# B&R Automation Studio project ControlPLC_DataDistribution (part 2)

### IoMap.iom - 5PC900_TS17_02/IoMap.iom
```iecst
VAR_CONFIG
	::VFLCR_Ope0:IO.raw.oSystemControl AT %QD."VF-LCR".SYSTEM_CONTROL_I2004Out;
	::VFLCR_Ope0:IO.ao.SelectedPrintNumber AT %QD."VF-LCR".SELECTED_PRINT_NUMBER_I200BOut;
	::VFLCR_Ope0:IO.ao.SelectedLayerNumber AT %QD."VF-LCR".SELECTED_LAYER_NUMBER_I200COut;
	::VFLCR_Ope0:IO.ao.SelectedBuildLayout AT %QD."VF-LCR".SELECTED_BUILD_LAYOUT_I200AOut;
	::VFLCR_Ope0:IO.ao.PLCHeartbeat AT %QD."VF-LCR".PLC_HEARTBEAT_I2003Out;
	::VFLCR_Ope0:IO.raw.oOperationControl AT %QD."VF-LCR".OPERATION_CONTROL_I2005Out;
	::VFLCR_Ope0:IO.raw.oManualLaserOperation AT %QD."VF-LCR".MANUAL_LASER_OPERATION_I200EOut;
	::VFLCR_Ope0:IO.raw.oManualLaserCurrentSetpoint AT %QD."VF-LCR".MANUAL_LASER_CURRENT_SETPOINT_I200FOut;
	::VFLCR_Ope0:IO.raw.oLaserEnable AT %QD."VF-LCR".LASER_ENABLE_I2008Out;
	::VFLCR_Ope0:IO.raw.oEnableLaserMainPower AT %QD."VF-LCR".LASER_REMOTE_START_I2010Out;
	::VFLCR_Ope0:IO.raw.oEnableLaserEmission AT %QD."VF-LCR".LASER_EMISSION_CONTROL_I2012Out;
	::VFLCR_Ope0:IO.raw.oEnableGuideLaser AT %QD."VF-LCR".GUIDE_LASER_CONTROL_I2011Out;
	::VFLCR_Ope0:IO.raw.oResetLaserErrors AT %QD."VF-LCR".LASER_RESET_I2013Out;
	::VFLCR_Ope0:IO.di.PowerlinkModuleOK AT %IX."VF-LCR".ModuleOk;
	::VFLCR_Ope0:IO.ai.DMACurrentTrajectory[0] AT %ID."VF-LCR".Entry_I201B_S01;
	::VFLCR_Ope0:IO.raw.iLaserFatalError AT %ID."VF-LCR".SYSTEM_ERROR_I2018;
	::VFLCR_Ope0:IO.raw.iSystemStatus AT %ID."VF-LCR".SYSTEM_STATUS_I2006;
	::VFLCR_Ope0:IO.ai.SystemHeartbeat AT %ID."VF-LCR".SYSTEM_HEARTBEAT_I2002;
	::VFLCR_Ope0:IO.raw.iSoftwareRevision AT %ID."VF-LCR".SOFTWARE_REVISION_I201D;
	::VFLCR_Ope0:IO.raw.iOperationStatus AT %ID."VF-LCR".OPERATION_STATUS_I2007;
	::VFLCR_Ope0:IO.raw.iManualModeLaserPower AT %ID."VF-LCR".LASER_POWER_MONITOR_I2019;
	::VFLCR_Ope0:IO.ai.LUTFiles_CalibrationID AT %ID."VF-LCR".LUT_LOAD_STATUS_I2009;
	::VFLCR_Ope0:IO.raw.iLaserWatchdogError AT %ID."VF-LCR".LASER_WATCHDOG_ERROR_I201E;
	::VFLCR_Ope0:IO.raw.iLaserEmissionEnabled AT %ID."VF-LCR".LASER_EMISSION_ON_I2017;
	::VFLCR_Ope0:IO.raw.iLaserControlPowerEnabled AT %ID."VF-LCR".LASER_CONTROL_SYSTEM_POWERED_ON_I2015;
	::VFLCR_Ope0:IO.raw.iFPGARevision AT %ID."VF-LCR".FPGA_REVISION_I2001;
	::VFLCR_Ope0:IO.ai.DMAStatus[8] AT %ID."VF-LCR".Entry_I201A_S09;
	::VFLCR_Ope0:IO.ai.DMAStatus[7] AT %ID."VF-LCR".Entry_I201A_S08;
	::VFLCR_Ope0:IO.ai.DMAStatus[6] AT %ID."VF-LCR".Entry_I201A_S07;
	::VFLCR_Ope0:IO.ai.DMAStatus[5] AT %ID."VF-LCR".Entry_I201A_S06;
	::VFLCR_Ope0:IO.ai.DMAStatus[4] AT %ID."VF-LCR".Entry_I201A_S05;
	::VFLCR_Ope0:IO.ai.DMAStatus[3] AT %ID."VF-LCR".Entry_I201A_S04;
	::VFLCR_Ope0:IO.ai.DMAStatus[13] AT %ID."VF-LCR".Entry_I201A_S0E;
	::VFLCR_Ope0:IO.ai.DMAStatus[2] AT %ID."VF-LCR".Entry_I201A_S03;
	::VFLCR_Ope0:IO.ai.DMAStatus[19] AT %ID."VF-LCR".Entry_I201A_S14;
	::VFLCR_Ope0:IO.ai.DMAStatus[1] AT %ID."VF-LCR".Entry_I201A_S02;
	::VFLCR_Ope0:IO.ai.DMAStatus[18] AT %ID."VF-LCR".Entry_I201A_S13;
	::VFLCR_Ope0:IO.ai.DMAStatus[17] AT %ID."VF-LCR".Entry_I201A_S12;
	::VFLCR_Ope0:IO.ai.DMAStatus[16] AT %ID."VF-LCR".Entry_I201A_S11;
	::VFLCR_Ope0:IO.ai.DMAStatus[15] AT %ID."VF-LCR".Entry_I201A_S10;
	::VFLCR_Ope0:IO.ai.DMAStatus[14] AT %ID."VF-LCR".Entry_I201A_S0F;
	::VFLCR_Ope0:IO.raw.iLaserMainPowerEnabled AT %ID."VF-LCR".LASER_MAIN_POWER_ON_I2016;
	::VFLCR_Ope0:IO.raw.iLaserReady_Error AT %ID."VF-LCR".LASER_ERROR_READY_I2014;
	::VFLCR_Ope0:IO.ai.DMAStatus[20] AT %ID."VF-LCR".Entry_I201A_S15;
	::VFLCR_Ope0:IO.ai.DMAStatus[12] AT %ID."VF-LCR".Entry_I201A_S0D;
	::VFLCR_Ope0:IO.ai.DMACurrentTrajectory[7] AT %ID."VF-LCR".Entry_I201B_S08;
	::VFLCR_Ope0:IO.ai.DMAStatus[0] AT %ID."VF-LCR".Entry_I201A_S01;
	::VFLCR_Ope0:IO.ai.DMALastPacketPosition[8] AT %ID."VF-LCR".Entry_I201C_S09;
	::VFLCR_Ope0:IO.ai.DMALastPacketPosition[7] AT %ID."VF-LCR".Entry_I201C_S08;
	::VFLCR_Ope0:IO.ai.DMALastPacketPosition[6] AT %ID."VF-LCR".Entry_I201C_S07;
	::VFLCR_Ope0:IO.ai.DMALastPacketPosition[5] AT %ID."VF-LCR".Entry_I201C_S06;
	::VFLCR_Ope0:IO.ai.DMALastPacketPosition[4] AT %ID."VF-LCR".Entry_I201C_S05;
	::VFLCR_Ope0:IO.ai.DMALastPacketPosition[3] AT %ID."VF-LCR".Entry_I201C_S04;
	::VFLCR_Ope0:IO.ai.DMALastPacketPosition[2] AT %ID."VF-LCR".Entry_I201C_S03;
	::VFLCR_Ope0:IO.ai.DMALastPacketPosition[19] AT %ID."VF-LCR".Entry_I201C_S14;
	::VFLCR_Ope0:IO.ai.DMAStatus[9] AT %ID."VF-LCR".Entry_I201A_S0A;
	::VFLCR_Ope0:IO.ai.DMALastPacketPosition[20] AT %ID."VF-LCR".Entry_I201C_S15;
	::VFLCR_Ope0:IO.ai.DMALastPacketPosition[18] AT %ID."VF-LCR".Entry_I201C_S13;
	::VFLCR_Ope0:IO.ai.DMALastPacketPosition[17] AT %ID."VF-LCR".Entry_I201C_S12;
	::VFLCR_Ope0:IO.ai.DMALastPacketPosition[16] AT %ID."VF-LCR".Entry_I201C_S11;
	::VFLCR_Ope0:IO.ai.DMALastPacketPosition[15] AT %ID."VF-LCR".Entry_I201C_S10;
	::VFLCR_Ope0:IO.ai.DMALastPacketPosition[14] AT %ID."VF-LCR".Entry_I201C_S0F;
	::VFLCR_Ope0:IO.ai.DMALastPacketPosition[13] AT %ID."VF-LCR".Entry_I201C_S0E;
	::VFLCR_Ope0:IO.ai.DMALastPacketPosition[12] AT %ID."VF-LCR".Entry_I201C_S0D;
	::VFLCR_Ope0:IO.ai.DMALastPacketPosition[11] AT %ID."VF-LCR".Entry_I201C_S0C;
	::VFLCR_Ope0:IO.ai.DMAStatus[10] AT %ID."VF-LCR".Entry_I201A_S0B;
	::VFLCR_Ope0:IO.ai.DMALastPacketPosition[1] AT %ID."VF-LCR".Entry_I201C_S02;
	::VFLCR_Ope0:IO.ai.DMAStatus[11] AT %ID."VF-LCR".Entry_I201A_S0C;
	::VFLCR_Ope0:IO.ai.DMALastPacketPosition[10] AT %ID."VF-LCR".Entry_I201C_S0B;
	::VFLCR_Ope0:IO.ai.DMALastPacketPosition[0] AT %ID."VF-LCR".Entry_I201C_S01;
	::VFLCR_Ope0:IO.ai.DMACurrentTrajectory[6] AT %ID."VF-LCR".Entry_I201B_S07;
	::VFLCR_Ope0:IO.ai.DMACurrentTrajectory[5] AT %ID."VF-LCR".Entry_I201B_S06;
	::VFLCR_Ope0:IO.ai.DMACurrentTrajectory[4] AT %ID."VF-LCR".Entry_I201B_S05;
	::VFLCR_Ope0:IO.ai.DMACurrentTrajectory[3] AT %ID."VF-LCR".Entry_I201B_S04;
	::VFLCR_Ope0:IO.ai.DMACurrentTrajectory[2] AT %ID."VF-LCR".Entry_I201B_S03;
	::VFLCR_Ope0:IO.ai.DMACurrentTrajectory[20] AT %ID."VF-LCR".Entry_I201B_S15;
	::VFLCR_Ope0:IO.ai.DMACurrentTrajectory[19] AT %ID."VF-LCR".Entry_I201B_S14;
	::VFLCR_Ope0:IO.ai.DMACurrentTrajectory[1] AT %ID."VF-LCR".Entry_I201B_S02;
	::VFLCR_Ope0:IO.ai.DMACurrentTrajectory[18] AT %ID."VF-LCR".Entry_I201B_S13;
	::VFLCR_Ope0:IO.ai.DMALastPacketPosition[9] AT %ID."VF-LCR".Entry_I201C_S0A;
	::VFLCR_Ope0:IO.ai.DMACurrentTrajectory[17] AT %ID."VF-LCR".Entry_I201B_S12;
	::VFLCR_Ope0:IO.ai.DMACurrentTrajectory[15] AT %ID."VF-LCR".Entry_I201B_S10;
	::VFLCR_Ope0:IO.ai.DMACurrentTrajectory[14] AT %ID."VF-LCR".Entry_I201B_S0F;
	::VFLCR_Ope0:IO.ai.DMACurrentTrajectory[13] AT %ID."VF-LCR".Entry_I201B_S0E;
	::VFLCR_Ope0:IO.ai.DMACurrentTrajectory[12] AT %ID."VF-LCR".Entry_I201B_S0D;
	::VFLCR_Ope0:IO.ai.DMACurrentTrajectory[11] AT %ID."VF-LCR".Entry_I201B_S0C;
	::VFLCR_Ope0:IO.ai.DMACurrentTrajectory[10] AT %ID."VF-LCR".Entry_I201B_S0B;
	::VFLCR_Ope0:IO.ai.DMACurrentTrajectory[9] AT %ID."VF-LCR".Entry_I201B_S0A;
	::VFLCR_Ope0:IO.ai.DMACurrentTrajectory[8] AT %ID."VF-LCR".Entry_I201B_S09;
	::VFLCR_Ope0:IO.ai.DMACurrentTrajectory[16] AT %ID."VF-LCR".Entry_I201B_S11;
	::VFLCR_Ope1:IO.raw.oSystemControl AT %QD."VF-LCR1".SYSTEM_CONTROL_I2004Out;
	::VFLCR_Ope1:IO.ao.SelectedPrintNumber AT %QD."VF-LCR1".SELECTED_PRINT_NUMBER_I200BOut;
	::VFLCR_Ope1:IO.ao.SelectedLayerNumber AT %QD."VF-LCR1".SELECTED_LAYER_NUMBER_I200COut;
	::VFLCR_Ope1:IO.ao.SelectedBuildLayout AT %QD."VF-LCR1".SELECTED_BUILD_LAYOUT_I200AOut;
	::VFLCR_Ope1:IO.ao.PLCHeartbeat AT %QD."VF-LCR1".PLC_HEARTBEAT_I2003Out;
	::VFLCR_Ope1:IO.raw.oOperationControl AT %QD."VF-LCR1".OPERATION_CONTROL_I2005Out;
	::VFLCR_Ope1:IO.raw.oManualLaserOperation AT %QD."VF-LCR1".MANUAL_LASER_OPERATION_I200EOut;
	::VFLCR_Ope1:IO.raw.oManualLaserCurrentSetpoint AT %QD."VF-LCR1".MANUAL_LASER_CURRENT_SETPOINT_I200FOut;
	::VFLCR_Ope1:IO.raw.oLaserEnable AT %QD."VF-LCR1".LASER_ENABLE_I2008Out;
	::VFLCR_Ope1:IO.raw.oEnableLaserMainPower AT %QD."VF-LCR1".LASER_REMOTE_START_I2010Out;
	::VFLCR_Ope1:IO.raw.oEnableLaserEmission AT %QD."VF-LCR1".LASER_EMISSION_CONTROL_I2012Out;
	::VFLCR_Ope1:IO.raw.oEnableGuideLaser AT %QD."VF-LCR1".GUIDE_LASER_CONTROL_I2011Out;
	::VFLCR_Ope1:IO.raw.oResetLaserErrors AT %QD."VF-LCR1".LASER_RESET_I2013Out;
	::VFLCR_Ope1:IO.di.PowerlinkModuleOK AT %IX."VF-LCR1".ModuleOk;
	::VFLCR_Ope1:IO.ai.DMACurrentTrajectory[0] AT %ID."VF-LCR1".Entry_I201B_S01;
	::VFLCR_Ope1:IO.raw.iLaserFatalError AT %ID."VF-LCR1".SYSTEM_ERROR_I2018;
	::VFLCR_Ope1:IO.raw.iSystemStatus AT %ID."VF-LCR1".SYSTEM_STATUS_I2006;
	::VFLCR_Ope1:IO.ai.SystemHeartbeat AT %ID."VF-LCR1".SYSTEM_HEARTBEAT_I2002;
	::VFLCR_Ope1:IO.raw.iSoftwareRevision AT %ID."VF-LCR1".SOFTWARE_REVISION_I201D;
	::VFLCR_Ope1:IO.raw.iOperationStatus AT %ID."VF-LCR1".OPERATION_STATUS_I2007;
	::VFLCR_Ope1:IO.raw.iManualModeLaserPower AT %ID."VF-LCR1".LASER_POWER_MONITOR_I2019;
	::VFLCR_Ope1:IO.ai.LUTFiles_CalibrationID AT %ID."VF-LCR1".LUT_LOAD_STATUS_I2009;
	::VFLCR_Ope1:IO.raw.iLaserWatchdogError AT %ID."VF-LCR1".LASER_WATCHDOG_ERROR_I201E;
	::VFLCR_Ope1:IO.raw.iLaserEmissionEnabled AT %ID."VF-LCR1".LASER_EMISSION_ON_I2017;
	::VFLCR_Ope1:IO.raw.iLaserControlPowerEnabled AT %ID."VF-LCR1".LASER_CONTROL_SYSTEM_POWERED_ON_I2015;
	::VFLCR_Ope1:IO.raw.iFPGARevision AT %ID."VF-LCR1".FPGA_REVISION_I2001;
	::VFLCR_Ope1:IO.ai.DMAStatus[8] AT %ID."VF-LCR1".Entry_I201A_S09;
	::VFLCR_Ope1:IO.ai.DMAStatus[7] AT %ID."VF-LCR1".Entry_I201A_S08;
	::VFLCR_Ope1:IO.ai.DMAStatus[6] AT %ID."VF-LCR1".Entry_I201A_S07;
	::VFLCR_Ope1:IO.ai.DMAStatus[5] AT %ID."VF-LCR1".Entry_I201A_S06;
	::VFLCR_Ope1:IO.ai.DMAStatus[4] AT %ID."VF-LCR1".Entry_I201A_S05;
	::VFLCR_Ope1:IO.ai.DMAStatus[3] AT %ID."VF-LCR1".Entry_I201A_S04;
	::VFLCR_Ope1:IO.ai.DMAStatus[13] AT %ID."VF-LCR1".Entry_I201A_S0E;
	::VFLCR_Ope1:IO.ai.DMAStatus[2] AT %ID."VF-LCR1".Entry_I201A_S03;
	::VFLCR_Ope1:IO.ai.DMAStatus[19] AT %ID."VF-LCR1".Entry_I201A_S14;
	::VFLCR_Ope1:IO.ai.DMAStatus[1] AT %ID."VF-LCR1".Entry_I201A_S02;
	::VFLCR_Ope1:IO.ai.DMAStatus[18] AT %ID."VF-LCR1".Entry_I201A_S13;
	::VFLCR_Ope1:IO.ai.DMAStatus[17] AT %ID."VF-LCR1".Entry_I201A_S12;
	::VFLCR_Ope1:IO.ai.DMAStatus[16] AT %ID."VF-LCR1".Entry_I201A_S11;
	::VFLCR_Ope1:IO.ai.DMAStatus[15] AT %ID."VF-LCR1".Entry_I201A_S10;
	::VFLCR_Ope1:IO.ai.DMAStatus[14] AT %ID."VF-LCR1".Entry_I201A_S0F;
	::VFLCR_Ope1:IO.raw.iLaserMainPowerEnabled AT %ID."VF-LCR1".LASER_MAIN_POWER_ON_I2016;
	::VFLCR_Ope1:IO.raw.iLaserReady_Error AT %ID."VF-LCR1".LASER_ERROR_READY_I2014;
	::VFLCR_Ope1:IO.ai.DMAStatus[20] AT %ID."VF-LCR1".Entry_I201A_S15;
	::VFLCR_Ope1:IO.ai.DMAStatus[12] AT %ID."VF-LCR1".Entry_I201A_S0D;
	::VFLCR_Ope1:IO.ai.DMACurrentTrajectory[7] AT %ID."VF-LCR1".Entry_I201B_S08;
	::VFLCR_Ope1:IO.ai.DMAStatus[0] AT %ID."VF-LCR1".Entry_I201A_S01;
	::VFLCR_Ope1:IO.ai.DMALastPacketPosition[8] AT %ID."VF-LCR1".Entry_I201C_S09;
	::VFLCR_Ope1:IO.ai.DMALastPacketPosition[7] AT %ID."VF-LCR1".Entry_I201C_S08;
	::VFLCR_Ope1:IO.ai.DMALastPacketPosition[6] AT %ID."VF-LCR1".Entry_I201C_S07;
	::VFLCR_Ope1:IO.ai.DMALastPacketPosition[5] AT %ID."VF-LCR1".Entry_I201C_S06;
	::VFLCR_Ope1:IO.ai.DMALastPacketPosition[4] AT %ID."VF-LCR1".Entry_I201C_S05;
	::VFLCR_Ope1:IO.ai.DMALastPacketPosition[3] AT %ID."VF-LCR1".Entry_I201C_S04;
	::VFLCR_Ope1:IO.ai.DMALastPacketPosition[2] AT %ID."VF-LCR1".Entry_I201C_S03;
	::VFLCR_Ope1:IO.ai.DMALastPacketPosition[19] AT %ID."VF-LCR1".Entry_I201C_S14;
	::VFLCR_Ope1:IO.ai.DMAStatus[9] AT %ID."VF-LCR1".Entry_I201A_S0A;
	::VFLCR_Ope1:IO.ai.DMALastPacketPosition[20] AT %ID."VF-LCR1".Entry_I201C_S15;
	::VFLCR_Ope1:IO.ai.DMALastPacketPosition[18] AT %ID."VF-LCR1".Entry_I201C_S13;
	::VFLCR_Ope1:IO.ai.DMALastPacketPosition[17] AT %ID."VF-LCR1".Entry_I201C_S12;
	::VFLCR_Ope1:IO.ai.DMALastPacketPosition[16] AT %ID."VF-LCR1".Entry_I201C_S11;
	::VFLCR_Ope1:IO.ai.DMALastPacketPosition[15] AT %ID."VF-LCR1".Entry_I201C_S10;
	::VFLCR_Ope1:IO.ai.DMALastPacketPosition[14] AT %ID."VF-LCR1".Entry_I201C_S0F;
	::VFLCR_Ope1:IO.ai.DMALastPacketPosition[13] AT %ID."VF-LCR1".Entry_I201C_S0E;
	::VFLCR_Ope1:IO.ai.DMALastPacketPosition[12] AT %ID."VF-LCR1".Entry_I201C_S0D;
	::VFLCR_Ope1:IO.ai.DMALastPacketPosition[11] AT %ID."VF-LCR1".Entry_I201C_S0C;
	::VFLCR_Ope1:IO.ai.DMAStatus[10] AT %ID."VF-LCR1".Entry_I201A_S0B;
	::VFLCR_Ope1:IO.ai.DMALastPacketPosition[1] AT %ID."VF-LCR1".Entry_I201C_S02;
	::VFLCR_Ope1:IO.ai.DMAStatus[11] AT %ID."VF-LCR1".Entry_I201A_S0C;
	::VFLCR_Ope1:IO.ai.DMALastPacketPosition[10] AT %ID."VF-LCR1".Entry_I201C_S0B;
	::VFLCR_Ope1:IO.ai.DMALastPacketPosition[0] AT %ID."VF-LCR1".Entry_I201C_S01;
	::VFLCR_Ope1:IO.ai.DMACurrentTrajectory[6] AT %ID."VF-LCR1".Entry_I201B_S07;
	::VFLCR_Ope1:IO.ai.DMACurrentTrajectory[5] AT %ID."VF-LCR1".Entry_I201B_S06;
	::VFLCR_Ope1:IO.ai.DMACurrentTrajectory[4] AT %ID."VF-LCR1".Entry_I201B_S05;
	::VFLCR_Ope1:IO.ai.DMACurrentTrajectory[3] AT %ID."VF-LCR1".Entry_I201B_S04;
	::VFLCR_Ope1:IO.ai.DMACurrentTrajectory[2] AT %ID."VF-LCR1".Entry_I201B_S03;
	::VFLCR_Ope1:IO.ai.DMACurrentTrajectory[20] AT %ID."VF-LCR1".Entry_I201B_S15;
	::VFLCR_Ope1:IO.ai.DMACurrentTrajectory[19] AT %ID."VF-LCR1".Entry_I201B_S14;
	::VFLCR_Ope1:IO.ai.DMACurrentTrajectory[1] AT %ID."VF-LCR1".Entry_I201B_S02;
	::VFLCR_Ope1:IO.ai.DMACurrentTrajectory[18] AT %ID."VF-LCR1".Entry_I201B_S13;
	::VFLCR_Ope1:IO.ai.DMALastPacketPosition[9] AT %ID."VF-LCR1".Entry_I201C_S0A;
	::VFLCR_Ope1:IO.ai.DMACurrentTrajectory[17] AT %ID."VF-LCR1".Entry_I201B_S12;
	::VFLCR_Ope1:IO.ai.DMACurrentTrajectory[15] AT %ID."VF-LCR1".Entry_I201B_S10;
	::VFLCR_Ope1:IO.ai.DMACurrentTrajectory[14] AT %ID."VF-LCR1".Entry_I201B_S0F;
	::VFLCR_Ope1:IO.ai.DMACurrentTrajectory[13] AT %ID."VF-LCR1".Entry_I201B_S0E;
	::VFLCR_Ope1:IO.ai.DMACurrentTrajectory[12] AT %ID."VF-LCR1".Entry_I201B_S0D;
	::VFLCR_Ope1:IO.ai.DMACurrentTrajectory[11] AT %ID."VF-LCR1".Entry_I201B_S0C;
	::VFLCR_Ope1:IO.ai.DMACurrentTrajectory[10] AT %ID."VF-LCR1".Entry_I201B_S0B;
	::VFLCR_Ope1:IO.ai.DMACurrentTrajectory[9] AT %ID."VF-LCR1".Entry_I201B_S0A;
	::VFLCR_Ope1:IO.ai.DMACurrentTrajectory[8] AT %ID."VF-LCR1".Entry_I201B_S09;
	::VFLCR_Ope1:IO.ai.DMACurrentTrajectory[16] AT %ID."VF-LCR1".Entry_I201B_S11;
	::VFLCR_Ope2:IO.raw.oSystemControl AT %QD."VF-LCR2".SYSTEM_CONTROL_I2004Out;
	::VFLCR_Ope2:IO.ao.SelectedPrintNumber AT %QD."VF-LCR2".SELECTED_PRINT_NUMBER_I200BOut;
	::VFLCR_Ope2:IO.ao.SelectedLayerNumber AT %QD."VF-LCR2".SELECTED_LAYER_NUMBER_I200COut;
	::VFLCR_Ope2:IO.ao.SelectedBuildLayout AT %QD."VF-LCR2".SELECTED_BUILD_LAYOUT_I200AOut;
	::VFLCR_Ope2:IO.ao.PLCHeartbeat AT %QD."VF-LCR2".PLC_HEARTBEAT_I2003Out;
	::VFLCR_Ope2:IO.raw.oOperationControl AT %QD."VF-LCR2".OPERATION_CONTROL_I2005Out;
	::VFLCR_Ope2:IO.raw.oManualLaserOperation AT %QD."VF-LCR2".MANUAL_LASER_OPERATION_I200EOut;
	::VFLCR_Ope2:IO.raw.oManualLaserCurrentSetpoint AT %QD."VF-LCR2".MANUAL_LASER_CURRENT_SETPOINT_I200FOut;
	::VFLCR_Ope2:IO.raw.oLaserEnable AT %QD."VF-LCR2".LASER_ENABLE_I2008Out;
	::VFLCR_Ope2:IO.raw.oEnableLaserMainPower AT %QD."VF-LCR2".LASER_REMOTE_START_I2010Out;
	::VFLCR_Ope2:IO.raw.oEnableLaserEmission AT %QD."VF-LCR2".LASER_EMISSION_CONTROL_I2012Out;
	::VFLCR_Ope2:IO.raw.oEnableGuideLaser AT %QD."VF-LCR2".GUIDE_LASER_CONTROL_I2011Out;
	::VFLCR_Ope2:IO.raw.oResetLaserErrors AT %QD."VF-LCR2".LASER_RESET_I2013Out;
	::VFLCR_Ope2:IO.di.PowerlinkModuleOK AT %IX."VF-LCR2".ModuleOk;
	::VFLCR_Ope2:IO.ai.DMACurrentTrajectory[0] AT %ID."VF-LCR2".Entry_I201B_S01;
	::VFLCR_Ope2:IO.raw.iLaserFatalError AT %ID."VF-LCR2".SYSTEM_ERROR_I2018;
	::VFLCR_Ope2:IO.raw.iSystemStatus AT %ID."VF-LCR2".SYSTEM_STATUS_I2006;
	::VFLCR_Ope2:IO.ai.SystemHeartbeat AT %ID."VF-LCR2".SYSTEM_HEARTBEAT_I2002;
	::VFLCR_Ope2:IO.raw.iSoftwareRevision AT %ID."VF-LCR2".SOFTWARE_REVISION_I201D;
	::VFLCR_Ope2:IO.raw.iOperationStatus AT %ID."VF-LCR2".OPERATION_STATUS_I2007;
	::VFLCR_Ope2:IO.raw.iManualModeLaserPower AT %ID."VF-LCR2".LASER_POWER_MONITOR_I2019;
	::VFLCR_Ope2:IO.ai.LUTFiles_CalibrationID AT %ID."VF-LCR2".LUT_LOAD_STATUS_I2009;
	::VFLCR_Ope2:IO.raw.iLaserWatchdogError AT %ID."VF-LCR2".LASER_WATCHDOG_ERROR_I201E;
	::VFLCR_Ope2:IO.raw.iLaserEmissionEnabled AT %ID."VF-LCR2".LASER_EMISSION_ON_I2017;
	::VFLCR_Ope2:IO.raw.iLaserControlPowerEnabled AT %ID."VF-LCR2".LASER_CONTROL_SYSTEM_POWERED_ON_I2015;
	::VFLCR_Ope2:IO.raw.iFPGARevision AT %ID."VF-LCR2".FPGA_REVISION_I2001;
	::VFLCR_Ope2:IO.ai.DMAStatus[8] AT %ID."VF-LCR2".Entry_I201A_S09;
	::VFLCR_Ope2:IO.ai.DMAStatus[7] AT %ID."VF-LCR2".Entry_I201A_S08;
	::VFLCR_Ope2:IO.ai.DMAStatus[6] AT %ID."VF-LCR2".Entry_I201A_S07;
	::VFLCR_Ope2:IO.ai.DMAStatus[5] AT %ID."VF-LCR2".Entry_I201A_S06;
	::VFLCR_Ope2:IO.ai.DMAStatus[4] AT %ID."VF-LCR2".Entry_I201A_S05;
	::VFLCR_Ope2:IO.ai.DMAStatus[3] AT %ID."VF-LCR2".Entry_I201A_S04;
	::VFLCR_Ope2:IO.ai.DMAStatus[13] AT %ID."VF-LCR2".Entry_I201A_S0E;
	::VFLCR_Ope2:IO.ai.DMAStatus[2] AT %ID."VF-LCR2".Entry_I201A_S03;
	::VFLCR_Ope2:IO.ai.DMAStatus[19] AT %ID."VF-LCR2".Entry_I201A_S14;
	::VFLCR_Ope2:IO.ai.DMAStatus[1] AT %ID."VF-LCR2".Entry_I201A_S02;
	::VFLCR_Ope2:IO.ai.DMAStatus[18] AT %ID."VF-LCR2".Entry_I201A_S13;
	::VFLCR_Ope2:IO.ai.DMAStatus[17] AT %ID."VF-LCR2".Entry_I201A_S12;
	::VFLCR_Ope2:IO.ai.DMAStatus[16] AT %ID."VF-LCR2".Entry_I201A_S11;
	::VFLCR_Ope2:IO.ai.DMAStatus[15] AT %ID."VF-LCR2".Entry_I201A_S10;
	::VFLCR_Ope2:IO.ai.DMAStatus[14] AT %ID."VF-LCR2".Entry_I201A_S0F;
	::VFLCR_Ope2:IO.raw.iLaserMainPowerEnabled AT %ID."VF-LCR2".LASER_MAIN_POWER_ON_I2016;
	::VFLCR_Ope2:IO.raw.iLaserReady_Error AT %ID."VF-LCR2".LASER_ERROR_READY_I2014;
	::VFLCR_Ope2:IO.ai.DMAStatus[20] AT %ID."VF-LCR2".Entry_I201A_S15;
	::VFLCR_Ope2:IO.ai.DMAStatus[12] AT %ID."VF-LCR2".Entry_I201A_S0D;
	::VFLCR_Ope2:IO.ai.DMACurrentTrajectory[7] AT %ID."VF-LCR2".Entry_I201B_S08;
	::VFLCR_Ope2:IO.ai.DMAStatus[0] AT %ID."VF-LCR2".Entry_I201A_S01;
	::VFLCR_Ope2:IO.ai.DMALastPacketPosition[8] AT %ID."VF-LCR2".Entry_I201C_S09;
	::VFLCR_Ope2:IO.ai.DMALastPacketPosition[7] AT %ID."VF-LCR2".Entry_I201C_S08;
	::VFLCR_Ope2:IO.ai.DMALastPacketPosition[6] AT %ID."VF-LCR2".Entry_I201C_S07;
	::VFLCR_Ope2:IO.ai.DMALastPacketPosition[5] AT %ID."VF-LCR2".Entry_I201C_S06;
	::VFLCR_Ope2:IO.ai.DMALastPacketPosition[4] AT %ID."VF-LCR2".Entry_I201C_S05;
	::VFLCR_Ope2:IO.ai.DMALastPacketPosition[3] AT %ID."VF-LCR2".Entry_I201C_S04;
	::VFLCR_Ope2:IO.ai.DMALastPacketPosition[2] AT %ID."VF-LCR2".Entry_I201C_S03;
	::VFLCR_Ope2:IO.ai.DMALastPacketPosition[19] AT %ID."VF-LCR2".Entry_I201C_S14;
	::VFLCR_Ope2:IO.ai.DMAStatus[9] AT %ID."VF-LCR2".Entry_I201A_S0A;
	::VFLCR_Ope2:IO.ai.DMALastPacketPosition[20] AT %ID."VF-LCR2".Entry_I201C_S15;
	::VFLCR_Ope2:IO.ai.DMALastPacketPosition[18] AT %ID."VF-LCR2".Entry_I201C_S13;
	::VFLCR_Ope2:IO.ai.DMALastPacketPosition[17] AT %ID."VF-LCR2".Entry_I201C_S12;
	::VFLCR_Ope2:IO.ai.DMALastPacketPosition[16] AT %ID."VF-LCR2".Entry_I201C_S11;
	::VFLCR_Ope2:IO.ai.DMALastPacketPosition[15] AT %ID."VF-LCR2".Entry_I201C_S10;
	::VFLCR_Ope2:IO.ai.DMALastPacketPosition[14] AT %ID."VF-LCR2".Entry_I201C_S0F;
	::VFLCR_Ope2:IO.ai.DMALastPacketPosition[13] AT %ID."VF-LCR2".Entry_I201C_S0E;
	::VFLCR_Ope2:IO.ai.DMALastPacketPosition[12] AT %ID."VF-LCR2".Entry_I201C_S0D;
	::VFLCR_Ope2:IO.ai.DMALastPacketPosition[11] AT %ID."VF-LCR2".Entry_I201C_S0C;
	::VFLCR_Ope2:IO.ai.DMAStatus[10] AT %ID."VF-LCR2".Entry_I201A_S0B;
	::VFLCR_Ope2:IO.ai.DMALastPacketPosition[1] AT %ID."VF-LCR2".Entry_I201C_S02;
	::VFLCR_Ope2:IO.ai.DMAStatus[11] AT %ID."VF-LCR2".Entry_I201A_S0C;
	::VFLCR_Ope2:IO.ai.DMALastPacketPosition[10] AT %ID."VF-LCR2".Entry_I201C_S0B;
	::VFLCR_Ope2:IO.ai.DMALastPacketPosition[0] AT %ID."VF-LCR2".Entry_I201C_S01;
	::VFLCR_Ope2:IO.ai.DMACurrentTrajectory[6] AT %ID."VF-LCR2".Entry_I201B_S07;
	::VFLCR_Ope2:IO.ai.DMACurrentTrajectory[5] AT %ID."VF-LCR2".Entry_I201B_S06;
	::VFLCR_Ope2:IO.ai.DMACurrentTrajectory[4] AT %ID."VF-LCR2".Entry_I201B_S05;
	::VFLCR_Ope2:IO.ai.DMACurrentTrajectory[3] AT %ID."VF-LCR2".Entry_I201B_S04;
	::VFLCR_Ope2:IO.ai.DMACurrentTrajectory[2] AT %ID."VF-LCR2".Entry_I201B_S03;
	::VFLCR_Ope2:IO.ai.DMACurrentTrajectory[20] AT %ID."VF-LCR2".Entry_I201B_S15;
	::VFLCR_Ope2:IO.ai.DMACurrentTrajectory[19] AT %ID."VF-LCR2".Entry_I201B_S14;
	::VFLCR_Ope2:IO.ai.DMACurrentTrajectory[1] AT %ID."VF-LCR2".Entry_I201B_S02;
	::VFLCR_Ope2:IO.ai.DMACurrentTrajectory[18] AT %ID."VF-LCR2".Entry_I201B_S13;
	::VFLCR_Ope2:IO.ai.DMALastPacketPosition[9] AT %ID."VF-LCR2".Entry_I201C_S0A;
	::VFLCR_Ope2:IO.ai.DMACurrentTrajectory[17] AT %ID."VF-LCR2".Entry_I201B_S12;
	::VFLCR_Ope2:IO.ai.DMACurrentTrajectory[15] AT %ID."VF-LCR2".Entry_I201B_S10;
	::VFLCR_Ope2:IO.ai.DMACurrentTrajectory[14] AT %ID."VF-LCR2".Entry_I201B_S0F;
	::VFLCR_Ope2:IO.ai.DMACurrentTrajectory[13] AT %ID."VF-LCR2".Entry_I201B_S0E;
	::VFLCR_Ope2:IO.ai.DMACurrentTrajectory[12] AT %ID."VF-LCR2".Entry_I201B_S0D;
	::VFLCR_Ope2:IO.ai.DMACurrentTrajectory[11] AT %ID."VF-LCR2".Entry_I201B_S0C;
	::VFLCR_Ope2:IO.ai.DMACurrentTrajectory[10] AT %ID."VF-LCR2".Entry_I201B_S0B;
	::VFLCR_Ope2:IO.ai.DMACurrentTrajectory[9] AT %ID."VF-LCR2".Entry_I201B_S0A;
	::VFLCR_Ope2:IO.ai.DMACurrentTrajectory[8] AT %ID."VF-LCR2".Entry_I201B_S09;
	::VFLCR_Ope2:IO.ai.DMACurrentTrajectory[16] AT %ID."VF-LCR2".Entry_I201B_S11;
	::VFLCR_Ope3:IO.raw.oSystemControl AT %QD."VF-LCR3".SYSTEM_CONTROL_I2004Out;
	::VFLCR_Ope3:IO.ao.SelectedPrintNumber AT %QD."VF-LCR3".SELECTED_PRINT_NUMBER_I200BOut;
	::VFLCR_Ope3:IO.ao.SelectedLayerNumber AT %QD."VF-LCR3".SELECTED_LAYER_NUMBER_I200COut;
	::VFLCR_Ope3:IO.ao.SelectedBuildLayout AT %QD."VF-LCR3".SELECTED_BUILD_LAYOUT_I200AOut;
	::VFLCR_Ope3:IO.ao.PLCHeartbeat AT %QD."VF-LCR3".PLC_HEARTBEAT_I2003Out;
	::VFLCR_Ope3:IO.raw.oOperationControl AT %QD."VF-LCR3".OPERATION_CONTROL_I2005Out;
	::VFLCR_Ope3:IO.raw.oManualLaserOperation AT %QD."VF-LCR3".MANUAL_LASER_OPERATION_I200EOut;
	::VFLCR_Ope3:IO.raw.oManualLaserCurrentSetpoint AT %QD."VF-LCR3".MANUAL_LASER_CURRENT_SETPOINT_I200FOut;
	::VFLCR_Ope3:IO.raw.oLaserEnable AT %QD."VF-LCR3".LASER_ENABLE_I2008Out;
	::VFLCR_Ope3:IO.raw.oEnableLaserMainPower AT %QD."VF-LCR3".LASER_REMOTE_START_I2010Out;
	::VFLCR_Ope3:IO.raw.oEnableLaserEmission AT %QD."VF-LCR3".LASER_EMISSION_CONTROL_I2012Out;
	::VFLCR_Ope3:IO.raw.oEnableGuideLaser AT %QD."VF-LCR3".GUIDE_LASER_CONTROL_I2011Out;
	::VFLCR_Ope3:IO.raw.oResetLaserErrors AT %QD."VF-LCR3".LASER_RESET_I2013Out;
	::VFLCR_Ope3:IO.di.PowerlinkModuleOK AT %IX."VF-LCR3".ModuleOk;
	::VFLCR_Ope3:IO.ai.DMACurrentTrajectory[0] AT %ID."VF-LCR3".Entry_I201B_S01;
	::VFLCR_Ope3:IO.raw.iLaserFatalError AT %ID."VF-LCR3".SYSTEM_ERROR_I2018;
	::VFLCR_Ope3:IO.raw.iSystemStatus AT %ID."VF-LCR3".SYSTEM_STATUS_I2006;
	::VFLCR_Ope3:IO.ai.SystemHeartbeat AT %ID."VF-LCR3".SYSTEM_HEARTBEAT_I2002;
	::VFLCR_Ope3:IO.raw.iSoftwareRevision AT %ID."VF-LCR3".SOFTWARE_REVISION_I201D;
	::VFLCR_Ope3:IO.raw.iOperationStatus AT %ID."VF-LCR3".OPERATION_STATUS_I2007;
	::VFLCR_Ope3:IO.raw.iManualModeLaserPower AT %ID."VF-LCR3".LASER_POWER_MONITOR_I2019;
	::VFLCR_Ope3:IO.ai.LUTFiles_CalibrationID AT %ID."VF-LCR3".LUT_LOAD_STATUS_I2009;
	::VFLCR_Ope3:IO.raw.iLaserWatchdogError AT %ID."VF-LCR3".LASER_WATCHDOG_ERROR_I201E;
	::VFLCR_Ope3:IO.raw.iLaserEmissionEnabled AT %ID."VF-LCR3".LASER_EMISSION_ON_I2017;
	::VFLCR_Ope3:IO.raw.iLaserControlPowerEnabled AT %ID."VF-LCR3".LASER_CONTROL_SYSTEM_POWERED_ON_I2015;
	::VFLCR_Ope3:IO.raw.iFPGARevision AT %ID."VF-LCR3".FPGA_REVISION_I2001;
	::VFLCR_Ope3:IO.ai.DMAStatus[8] AT %ID."VF-LCR3".Entry_I201A_S09;
	::VFLCR_Ope3:IO.ai.DMAStatus[7] AT %ID."VF-LCR3".Entry_I201A_S08;
	::VFLCR_Ope3:IO.ai.DMAStatus[6] AT %ID."VF-LCR3".Entry_I201A_S07;
	::VFLCR_Ope3:IO.ai.DMAStatus[5] AT %ID."VF-LCR3".Entry_I201A_S06;
	::VFLCR_Ope3:IO.ai.DMAStatus[4] AT %ID."VF-LCR3".Entry_I201A_S05;
	::VFLCR_Ope3:IO.ai.DMAStatus[3] AT %ID."VF-LCR3".Entry_I201A_S04;
	::VFLCR_Ope3:IO.ai.DMAStatus[13] AT %ID."VF-LCR3".Entry_I201A_S0E;
	::VFLCR_Ope3:IO.ai.DMAStatus[2] AT %ID."VF-LCR3".Entry_I201A_S03;
	::VFLCR_Ope3:IO.ai.DMAStatus[19] AT %ID."VF-LCR3".Entry_I201A_S14;
	::VFLCR_Ope3:IO.ai.DMAStatus[1] AT %ID."VF-LCR3".Entry_I201A_S02;
	::VFLCR_Ope3:IO.ai.DMAStatus[18] AT %ID."VF-LCR3".Entry_I201A_S13;
	::VFLCR_Ope3:IO.ai.DMAStatus[17] AT %ID."VF-LCR3".Entry_I201A_S12;
	::VFLCR_Ope3:IO.ai.DMAStatus[16] AT %ID."VF-LCR3".Entry_I201A_S11;
	::VFLCR_Ope3:IO.ai.DMAStatus[15] AT %ID."VF-LCR3".Entry_I201A_S10;
	::VFLCR_Ope3:IO.ai.DMAStatus[14] AT %ID."VF-LCR3".Entry_I201A_S0F;
	::VFLCR_Ope3:IO.raw.iLaserMainPowerEnabled AT %ID."VF-LCR3".LASER_MAIN_POWER_ON_I2016;
	::VFLCR_Ope3:IO.raw.iLaserReady_Error AT %ID."VF-LCR3".LASER_ERROR_READY_I2014;
	::VFLCR_Ope3:IO.ai.DMAStatus[20] AT %ID."VF-LCR3".Entry_I201A_S15;
	::VFLCR_Ope3:IO.ai.DMAStatus[12] AT %ID."VF-LCR3".Entry_I201A_S0D;
	::VFLCR_Ope3:IO.ai.DMACurrentTrajectory[7] AT %ID."VF-LCR3".Entry_I201B_S08;
	::VFLCR_Ope3:IO.ai.DMAStatus[0] AT %ID."VF-LCR3".Entry_I201A_S01;
	::VFLCR_Ope3:IO.ai.DMALastPacketPosition[8] AT %ID."VF-LCR3".Entry_I201C_S09;
	::VFLCR_Ope3:IO.ai.DMALastPacketPosition[7] AT %ID."VF-LCR3".Entry_I201C_S08;
	::VFLCR_Ope3:IO.ai.DMALastPacketPosition[6] AT %ID."VF-LCR3".Entry_I201C_S07;
	::VFLCR_Ope3:IO.ai.DMALastPacketPosition[5] AT %ID."VF-LCR3".Entry_I201C_S06;
	::VFLCR_Ope3:IO.ai.DMALastPacketPosition[4] AT %ID."VF-LCR3".Entry_I201C_S05;
	::VFLCR_Ope3:IO.ai.DMALastPacketPosition[3] AT %ID."VF-LCR3".Entry_I201C_S04;
	::VFLCR_Ope3:IO.ai.DMALastPacketPosition[2] AT %ID."VF-LCR3".Entry_I201C_S03;
	::VFLCR_Ope3:IO.ai.DMALastPacketPosition[19] AT %ID."VF-LCR3".Entry_I201C_S14;
	::VFLCR_Ope3:IO.ai.DMAStatus[9] AT %ID."VF-LCR3".Entry_I201A_S0A;
	::VFLCR_Ope3:IO.ai.DMALastPacketPosition[20] AT %ID."VF-LCR3".Entry_I201C_S15;
	::VFLCR_Ope3:IO.ai.DMALastPacketPosition[18] AT %ID."VF-LCR3".Entry_I201C_S13;
	::VFLCR_Ope3:IO.ai.DMALastPacketPosition[17] AT %ID."VF-LCR3".Entry_I201C_S12;
	::VFLCR_Ope3:IO.ai.DMALastPacketPosition[16] AT %ID."VF-LCR3".Entry_I201C_S11;
	::VFLCR_Ope3:IO.ai.DMALastPacketPosition[15] AT %ID."VF-LCR3".Entry_I201C_S10;
	::VFLCR_Ope3:IO.ai.DMALastPacketPosition[14] AT %ID."VF-LCR3".Entry_I201C_S0F;
	::VFLCR_Ope3:IO.ai.DMALastPacketPosition[13] AT %ID."VF-LCR3".Entry_I201C_S0E;
	::VFLCR_Ope3:IO.ai.DMALastPacketPosition[12] AT %ID."VF-LCR3".Entry_I201C_S0D;
	::VFLCR_Ope3:IO.ai.DMALastPacketPosition[11] AT %ID."VF-LCR3".Entry_I201C_S0C;
	::VFLCR_Ope3:IO.ai.DMAStatus[10] AT %ID."VF-LCR3".Entry_I201A_S0B;
	::VFLCR_Ope3:IO.ai.DMALastPacketPosition[1] AT %ID."VF-LCR3".Entry_I201C_S02;
	::VFLCR_Ope3:IO.ai.DMAStatus[11] AT %ID."VF-LCR3".Entry_I201A_S0C;
	::VFLCR_Ope3:IO.ai.DMALastPacketPosition[10] AT %ID."VF-LCR3".Entry_I201C_S0B;
	::VFLCR_Ope3:IO.ai.DMALastPacketPosition[0] AT %ID."VF-LCR3".Entry_I201C_S01;
	::VFLCR_Ope3:IO.ai.DMACurrentTrajectory[6] AT %ID."VF-LCR3".Entry_I201B_S07;
	::VFLCR_Ope3:IO.ai.DMACurrentTrajectory[5] AT %ID."VF-LCR3".Entry_I201B_S06;
	::VFLCR_Ope3:IO.ai.DMACurrentTrajectory[4] AT %ID."VF-LCR3".Entry_I201B_S05;
	::VFLCR_Ope3:IO.ai.DMACurrentTrajectory[3] AT %ID."VF-LCR3".Entry_I201B_S04;
	::VFLCR_Ope3:IO.ai.DMACurrentTrajectory[2] AT %ID."VF-LCR3".Entry_I201B_S03;
	::VFLCR_Ope3:IO.ai.DMACurrentTrajectory[20] AT %ID."VF-LCR3".Entry_I201B_S15;
	::VFLCR_Ope3:IO.ai.DMACurrentTrajectory[19] AT %ID."VF-LCR3".Entry_I201B_S14;
	::VFLCR_Ope3:IO.ai.DMACurrentTrajectory[1] AT %ID."VF-LCR3".Entry_I201B_S02;
	::VFLCR_Ope3:IO.ai.DMACurrentTrajectory[18] AT %ID."VF-LCR3".Entry_I201B_S13;
	::VFLCR_Ope3:IO.ai.DMALastPacketPosition[9] AT %ID."VF-LCR3".Entry_I201C_S0A;
	::VFLCR_Ope3:IO.ai.DMACurrentTrajectory[17] AT %ID."VF-LCR3".Entry_I201B_S12;
	::VFLCR_Ope3:IO.ai.DMACurrentTrajectory[15] AT %ID."VF-LCR3".Entry_I201B_S10;
	::VFLCR_Ope3:IO.ai.DMACurrentTrajectory[14] AT %ID."VF-LCR3".Entry_I201B_S0F;
	::VFLCR_Ope3:IO.ai.DMACurrentTrajectory[13] AT %ID."VF-LCR3".Entry_I201B_S0E;
	::VFLCR_Ope3:IO.ai.DMACurrentTrajectory[12] AT %ID."VF-LCR3".Entry_I201B_S0D;
	::VFLCR_Ope3:IO.ai.DMACurrentTrajectory[11] AT %ID."VF-LCR3".Entry_I201B_S0C;
	::VFLCR_Ope3:IO.ai.DMACurrentTrajectory[10] AT %ID."VF-LCR3".Entry_I201B_S0B;
	::VFLCR_Ope3:IO.ai.DMACurrentTrajectory[9] AT %ID."VF-LCR3".Entry_I201B_S0A;
	::VFLCR_Ope3:IO.ai.DMACurrentTrajectory[8] AT %ID."VF-LCR3".Entry_I201B_S09;
	::VFLCR_Ope3:IO.ai.DMACurrentTrajectory[16] AT %ID."VF-LCR3".Entry_I201B_S11;
	::Safety:IO.LaserSystem[0].SDI_RackPowerContactorB_EDM.CH1 AT %IX."CM402_SC_LaserRack1".SafeDigitalInput02;
	::Safety:IO.LaserSystem[0].SDI_VFLCR_SafetyRelayEDM.CH1 AT %IX."CM402_SC_LaserRack1".SafeDigitalInput03;
	::Safety:IO.LaserSystem[0].SDI_RackPowerContactorA_EDM.SAFEOK AT %IX."CM402_SC_LaserRack1".SafeInputOK01;
	::Safety:IO.LaserSystem[0].SDI_RackPowerContactorB_EDM.SAFEOK AT %IX."CM402_SC_LaserRack1".SafeInputOK02;
	::Safety:IO.LaserSystem[0].SDI_VFLCR_SafetyRelayEDM.SAFEOK AT %IX."CM402_SC_LaserRack1".SafeInputOK03;
	::Safety:IO.LaserSystem[0].SDO_RackPowerContactor.CH1 AT %IX."CM402_SC_LaserRack1".PhysicalStateOutput01;
	::Safety:IO.LaserSystem[0].SDO_RackPowerContactor.CH2 AT %IX."CM402_SC_LaserRack1".PhysicalStateOutput02;
	::Safety:IO.LaserSystem[0].SDO_RackPowerContactor.CH1_SAFEOK AT %IX."CM402_SC_LaserRack1".SafeOutputOK01;
	::Safety:IO.LaserSystem[0].SDO_RackPowerContactor.CH2_SAFEOK AT %IX."CM402_SC_LaserRack1".SafeOutputOK02;
	::Safety:IO.LaserSystem[0].SDO_VFLCR_SafetyRelay.CH1 AT %IX."CM402_SC_LaserRack1".PhysicalStateOutput03;
	::Safety:IO.LaserSystem[0].SDO_VFLCR_SafetyRelay.CH2 AT %IX."CM402_SC_LaserRack1".PhysicalStateOutput04;
	::Safety:IO.LaserSystem[0].SDO_VFLCR_SafetyRelay.CH1_SAFEOK AT %IX."CM402_SC_LaserRack1".SafeOutputOK03;
	::Safety:IO.LaserSystem[0].SDO_VFLCR_SafetyRelay.CH2_SAFEOK AT %IX."CM402_SC_LaserRack1".SafeOutputOK04;
	::Safety:IO.LaserSystem[0].SDI_RackPowerContactorA_EDM.CH1 AT %IX."CM402_SC_LaserRack1".SafeDigitalInput01;
	::Safety:IO.LaserSystem[1].SDI_RackPowerContactorA_EDM.CH1 AT %IX."CM403_SC_LaserRack2".SafeDigitalInput01;
	::Safety:IO.LaserSystem[1].SDI_RackPowerContactorB_EDM.CH1 AT %IX."CM403_SC_LaserRack2".SafeDigitalInput02;
	::Safety:IO.LaserSystem[1].SDI_VFLCR_SafetyRelayEDM.CH1 AT %IX."CM403_SC_LaserRack2".SafeDigitalInput03;
	::Safety:IO.LaserSystem[1].SDI_RackPowerContactorA_EDM.SAFEOK AT %IX."CM403_SC_LaserRack2".SafeInputOK01;
	::Safety:IO.LaserSystem[1].SDI_RackPowerContactorB_EDM.SAFEOK AT %IX."CM403_SC_LaserRack2".SafeInputOK02;
	::Safety:IO.LaserSystem[1].SDI_VFLCR_SafetyRelayEDM.SAFEOK AT %IX."CM403_SC_LaserRack2".SafeInputOK03;
	::Safety:IO.LaserSystem[1].SDO_RackPowerContactor.CH1_SAFEOK AT %IX."CM403_SC_LaserRack2".SafeOutputOK01;
	::Safety:IO.LaserSystem[1].SDO_RackPowerContactor.CH2_SAFEOK AT %IX."CM403_SC_LaserRack2".SafeOutputOK02;
	::Safety:IO.LaserSystem[1].SDO_RackPowerContactor.CH1 AT %IX."CM403_SC_LaserRack2".PhysicalStateOutput01;
	::Safety:IO.LaserSystem[1].SDO_RackPowerContactor.CH2 AT %IX."CM403_SC_LaserRack2".PhysicalStateOutput02;
	::Safety:IO.LaserSystem[1].SDO_VFLCR_SafetyRelay.CH1_SAFEOK AT %IX."CM403_SC_LaserRack2".SafeOutputOK03;
	::Safety:IO.LaserSystem[1].SDO_VFLCR_SafetyRelay.CH2_SAFEOK AT %IX."CM403_SC_LaserRack2".SafeOutputOK04;
	::Safety:IO.LaserSystem[1].SDO_VFLCR_SafetyRelay.CH1 AT %IX."CM403_SC_LaserRack2".PhysicalStateOutput03;
	::Safety:IO.LaserSystem[1].SDO_VFLCR_SafetyRelay.CH2 AT %IX."CM403_SC_LaserRack2".PhysicalStateOutput04;
	::Safety:IO.LaserSystem[2].SDI_RackPowerContactorA_EDM.CH1 AT %IX."CM404_SC_LaserRack3".SafeDigitalInput01;
	::Safety:IO.LaserSystem[2].SDI_RackPowerContactorB_EDM.CH1 AT %IX."CM404_SC_LaserRack3".SafeDigitalInput02;
	::Safety:IO.LaserSystem[2].SDI_VFLCR_SafetyRelayEDM.CH1 AT %IX."CM404_SC_LaserRack3".SafeDigitalInput03;
	::Safety:IO.LaserSystem[2].SDI_RackPowerContactorA_EDM.SAFEOK AT %IX."CM404_SC_LaserRack3".SafeInputOK01;
	::Safety:IO.LaserSystem[2].SDI_VFLCR_SafetyRelayEDM.SAFEOK AT %IX."CM404_SC_LaserRack3".SafeInputOK03;
	::Safety:IO.LaserSystem[2].SDO_RackPowerContactor.CH1 AT %IX."CM404_SC_LaserRack3".PhysicalStateOutput01;
	::Safety:IO.LaserSystem[2].SDO_RackPowerContactor.CH2 AT %IX."CM404_SC_LaserRack3".PhysicalStateOutput02;
	::Safety:IO.LaserSystem[2].SDO_RackPowerContactor.CH1_SAFEOK AT %IX."CM404_SC_LaserRack3".SafeOutputOK01;
	::Safety:IO.LaserSystem[2].SDO_RackPowerContactor.CH2_SAFEOK AT %IX."CM404_SC_LaserRack3".SafeOutputOK02;
	::Safety:IO.LaserSystem[2].SDO_VFLCR_SafetyRelay.CH1_SAFEOK AT %IX."CM404_SC_LaserRack3".SafeOutputOK03;
	::Safety:IO.LaserSystem[2].SDO_VFLCR_SafetyRelay.CH2_SAFEOK AT %IX."CM404_SC_LaserRack3".SafeOutputOK04;
	::Safety:IO.LaserSystem[2].SDO_VFLCR_SafetyRelay.CH1 AT %IX."CM404_SC_LaserRack3".PhysicalStateOutput03;
	::Safety:IO.LaserSystem[2].SDO_VFLCR_SafetyRelay.CH2 AT %IX."CM404_SC_LaserRack3".PhysicalStateOutput04;
	::Safety:IO.LaserSystem[3].SDI_RackPowerContactorA_EDM.CH1 AT %IX."CM405_SC_LaserRack4".SafeDigitalInput01;
	::Safety:IO.LaserSystem[3].SDI_RackPowerContactorB_EDM.CH1 AT %IX."CM405_SC_LaserRack4".SafeDigitalInput02;
	::Safety:IO.LaserSystem[3].SDI_VFLCR_SafetyRelayEDM.CH1 AT %IX."CM405_SC_LaserRack4".SafeDigitalInput03;
	::Safety:IO.LaserSystem[3].SDI_RackPowerContactorA_EDM.SAFEOK AT %IX."CM405_SC_LaserRack4".SafeInputOK01;
	::Safety:IO.LaserSystem[2].SDI_RackPowerContactorB_EDM.SAFEOK AT %IX."CM404_SC_LaserRack3".SafeInputOK02;
	::Safety:IO.LaserSystem[3].SDI_RackPowerContactorB_EDM.SAFEOK AT %IX."CM405_SC_LaserRack4".SafeInputOK02;
	::Safety:IO.LaserSystem[3].SDI_VFLCR_SafetyRelayEDM.SAFEOK AT %IX."CM405_SC_LaserRack4".SafeInputOK03;
	::Safety:IO.LaserSystem[3].SDO_RackPowerContactor.CH1_SAFEOK AT %IX."CM405_SC_LaserRack4".SafeOutputOK01;
	::Safety:IO.LaserSystem[3].SDO_RackPowerContactor.CH2_SAFEOK AT %IX."CM405_SC_LaserRack4".SafeOutputOK02;
	::Safety:IO.LaserSystem[3].SDO_VFLCR_SafetyRelay.CH1_SAFEOK AT %IX."CM405_SC_LaserRack4".SafeOutputOK03;
	::Safety:IO.LaserSystem[3].SDO_VFLCR_SafetyRelay.CH2_SAFEOK AT %IX."CM405_SC_LaserRack4".SafeOutputOK04;
	::Safety:IO.LaserSystem[3].SDO_RackPowerContactor.CH1 AT %IX."CM405_SC_LaserRack4".PhysicalStateOutput01;
	::Safety:IO.LaserSystem[3].SDO_RackPowerContactor.CH2 AT %IX."CM405_SC_LaserRack4".PhysicalStateOutput02;
	::Safety:IO.LaserSystem[3].SDO_VFLCR_SafetyRelay.CH1 AT %IX."CM405_SC_LaserRack4".PhysicalStateOutput03;
	::Safety:IO.LaserSystem[3].SDO_VFLCR_SafetyRelay.CH2 AT %IX."CM405_SC_LaserRack4".PhysicalStateOutput04;
	::Safety:IO.safeLOGIC.SafeModuleOK[10] AT %IX."CM402_SC_LaserRack1".SafeModuleOK;
	::Safety:IO.safeLOGIC.SafeModuleOK[11] AT %IX."CM403_SC_LaserRack2".SafeModuleOK;
	::Safety:IO.safeLOGIC.SafeModuleOK[12] AT %IX."CM404_SC_LaserRack3".SafeModuleOK;
	::Safety:IO.safeLOGIC.SafeModuleOK[13] AT %IX."CM405_SC_LaserRack4".SafeModuleOK;
	::Safety:IO.safeLOGIC.SafeModuleOK[0] AT %IX."X20SI8110".SafeModuleOK;
	::Safety:IO.SDI_EStopButton_ControlStation.DUAL_EVAL AT %IX."X20SI8110".SafeTwoChannelInput0102;
	::Safety:IO.SDI_EStopButton_SafetyLockoutBox.DUAL_EVAL AT %IX."X20SI8110".SafeTwoChannelInput0506;
	::Safety:IO.SDI_EStopButton_HandHeld.DUAL_EVAL AT %IX."X20SI8110".SafeTwoChannelInput0708;
	::Safety:IO.SDI_EStopButton_ControlStation.SAFEOK AT %IX."X20SI8110".SafeTwoChannelOK0102;
	::Safety:IO.SDI_EStopButton_SafetyLockoutBox.SAFEOK AT %IX."X20SI8110".SafeTwoChannelOK0506;
	::Safety:IO.SDI_EStopButton_HandHeld.SAFEOK AT %IX."X20SI8110".SafeTwoChannelOK0708;
	::Safety:IO.safeLOGIC.Command.RequestMachineSafetyReset AT %QX."X20SLX210".BOOL10001;
	::Safety:IO.safeLOGIC.Command.RequestLaserSafetyReset AT %QX."X20SLX210".BOOL10002;
	::Safety:IO.safeLOGIC.Command.RacksEnabled AT %QW."X20SLX210".UINT1001;
	::Safety:IO.safeLOGIC.Status.SafetySystemReady AT %IX."X20SLX210".BOOL00001;
	::Safety:IO.safeLOGIC.Status.SafetyReset_EStops AT %IX."X20SLX210".BOOL00002;
	::Safety:IO.safeLOGIC.Status.SafetyReset_Lasers AT %IX."X20SLX210".BOOL00005;
	::Safety:IO.safeLOGIC.Status.EStopPressed AT %IX."X20SLX210".BOOL00003;
	::Safety:IO.safeLOGIC.Status.SafetyProgramRevision AT %IW."X20SLX210".UINT0001;
	::Safety:IO.safeLOGIC.Command.EnableLaserSafetyInterlock AT %QX."X20SLX210".BOOL10003;
END_VAR
```

### MachineAC.mpalarmxcore - 5PC900_TS17_02/mappServices/MachineAC.mpalarmxcore
```
Element alarm_Machine (Type=mpalarmxcore)
  mapp.AlarmX.Core:
    Default:
      [0] = Reaction
Element alarm_Init (Type=mpalarmxcore)
Element alarm_Laser (Type=mpalarmxcore)
Element alarm_PermMem (Type=mpalarmxcore)
Element alarm_Safety (Type=mpalarmxcore)
Element alarm_MachineMode (Type=mpalarmxcore)
```

### MachineCG.mpcomgroup - 5PC900_TS17_02/mappServices/MachineCG.mpcomgroup
```
Element gGroup_Machine (Type=mpcomgroup)
  Linking:
    Subnodes:
      0 = alarm_Machine
      1 = gAlarmXHistory_Machine
      2 = gGroup_Init
      3 = gGroup_AxisBasic
      4 = gGroup_CncGantry
      5 = gGroup_Recoater
      6 = gGroup_Laser
      7 = gGroup_Vision
      8 = gGroup_Cooling
      9 = gGroup_Lift
      10 = gGroup_PrintMan
      11 = gGroup_Shuttle
      12 = gGroup_Pod
      13 = gGroup_Gas
      14 = gGroup_Pumps
      15 = gGroup_Filter
      16 = gGroup_Safety
      17 = gGroup_Leveling
      18 = gGroup_DataCollection
      19 = gGroup_Powder
      20 = gGroup_MachineMode
      21 = UserMgmtX
      22 = gUserXLogin
      23 = gGroup_Pod
Element gGroup_Pod (Type=mpcomgroup)
  Linking:
    Subnodes:
      0 = alarm_Pod
Element gGroup_Shuttle (Type=mpcomgroup)
  Linking:
    Subnodes:
      0 = alarm_Shuttle
      1 = gAxisShuttle
Element gGroup_Init (Type=mpcomgroup)
  Linking:
    Subnodes:
      0 = alarm_Init
Element gGroup_PrintMan (Type=mpcomgroup)
  Linking:
    Subnodes:
      0 = alarm_PrintMan
Element gGroup_AxisBasic (Type=mpcomgroup)
  Linking:
    Subnodes:
      0 = alarm_AxisBasic
Element gGroup_CncGantry (Type=mpcomgroup)
  Linking:
    Subnodes:
      0 = alarm_CncGantry
      1 = gCncGantry
      2 = gGroup_CncGear
Element gGroup_CncGear (Type=mpcomgroup)
  Linking:
    Subnodes:
      0 = alarm_GearSystemGantryX
      1 = gAxisGantryX1
      2 = gAxisGantryX2
Element gGroup_Recoater (Type=mpcomgroup)
  Linking:
    Subnodes:
      0 = alarm_Recoater
      1 = gAxisRecoater
      2 = gGroup_RecoaterGear
Element gGroup_RecoaterGear (Type=mpcomgroup)
  Linking:
    Subnodes:
      0 = alarm_GearSystemRecoaterX
      1 = gAxisRecoater1
      2 = gAxisRecoater2
Element gGroup_Lift (Type=mpcomgroup)
  Linking:
    Subnodes:
      0 = alarm_Lift
      1 = gAxisLiftZ
      2 = gGroup_LiftGear
      3 = gAxisLiftLinEnc1
      4 = gAxisLiftLinEnc2
      5 = gAxisLiftLinEnc3
Element gGroup_LiftGear (Type=mpcomgroup)
  Linking:
    Subnodes:
      0 = gAxisLiftZ1
      1 = gAxisLiftZ2
      2 = gAxisLiftZ3
      3 = alarm_GearSystemLiftZ
Element gGroup_Laser (Type=mpcomgroup)
  Linking:
    Subnodes:
      0 = alarm_Laser
Element gGroup_Cooling (Type=mpcomgroup)
  Linking:
    Subnodes:
      0 = alarm_Cooling
Element gGroup_Safety (Type=mpcomgroup)
  Linking:
    Subnodes:
      0 = alarm_Safety
Element gGroup_Gas (Type=mpcomgroup)
  Linking:
    Subnodes:
      0 = alarm_Gas
Element gGroup_Vision (Type=mpcomgroup)
  Linking:
    Subnodes:
      0 = alarm_Vision
Element gGroup_Pumps (Type=mpcomgroup)
  Linking:
    Subnodes:
      0 = alarm_Pumps
Element gGroup_Filter (Type=mpcomgroup)
  Linking:
    Subnodes:
      0 = alarm_Filter
Element gGroup_Leveling (Type=mpcomgroup)
  Linking:
    Subnodes:
      0 = alarm_Leveling
Element gGroup_MachineMode (Type=mpcomgroup)
  Linking:
    Subnodes:
      0 = alarm_MachineMode
Element gGroup_DataCollection (Type=mpcomgroup)
  Linking:
    Subnodes:
      0 = alarm_MQTT
Element gGroup_Powder (Type=mpcomgroup)
  Linking:
    Subnodes:
      0 = alarm_Powder
```

### Recipies.mprecipexml - 5PC900_TS17_02/mappServices/Recipies.mprecipexml
```
Element gBuildInfoRecipe (Type=mprecipexml)
  Alarms = MpAlarmX
    mapp.AlarmX.Core.Configuration:
      [0]:
        Code = 1300
        Severity = 4
        AdditionalInformation1 = Build Info
        AdditionalInformation2 = Recipe
      [1]:
        Code = 1301
        Severity = 4
        AdditionalInformation1 = Build Info
        AdditionalInformation2 = Recipe
      [2]:
        Code = 1302
        Severity = 4
        AdditionalInformation1 = Build Info
        AdditionalInformation2 = Recipe
      [3]:
        Code = 1303
        Severity = 4
        AdditionalInformation1 = Build Info
        AdditionalInformation2 = Recipe
```

## Logical view

Binary libraries used (declarations not repeated): operator, runtime, astime, AsIecCon, AsZip, FileIO, AsGuard, AsIODiag, sys_lib, AsBrStr, standard, AsArLog, ArEventLog, AsHttp, AsBrWStr, AsTCP, AsXml, LoopConR, AsBrMath, LoopCont, MTTypes, brsystem, McBase, McPathGen 5.19.3, MpAxis 5.19.3, McPureVAx 5.19.3, McAcpAx 5.19.3, McAxis 5.19.3, McProgInt 5.19.3, McAxGroup 5.19.3, MpBase, MpCnc 5.19.3, SfDomain, MpAlarmX, MpCom 5.19.0, MpRecipe 5.19.0, MTData 5.19.0, CoTrace, MTLookUp 5.19.0, AsIoTime, AsARCfg, MpWebXs 5.19.0, AsArSdm, MpUserX 5.19.0, IotMqtt, piper, fiowrap, messagebox 0.01.3, ringbuflib, hmitools, logthat, bodyguard, stringext 0.14.3, tcpcomm 0.10.0, databuffer 0.01.1, Finder 0.00.1, hammers 0.08.0, atn 0.04.6, AxisLib 4.02.0, omjson 1.03.8, csvfilelib, persist, vartools, ArCert, AsHW, AsETH, MTBasics

### Global.typ - Global data types
```iecst
TYPE
	Machine_typ : 	STRUCT
		operation : MACHINE_OPERATIONS_ENUM;
		_previousOperation : MACHINE_OPERATIONS_ENUM;
	END_STRUCT;
	MACHINE_OPERATIONS_ENUM :
		(
		MACH_OP_NONE,
		MACH_OP_START_DISTRIBUTION,
		MACH_OP_ABORT_DISTRIBUTION
		);
	SYSTEM_GENERAL_STATUS_ENUM :
		(
		PRINT_JOB_MANAGER_ERROR,
		BUILD_DISTRIBUTOR_ERROR,
		VFLCR_ERROR
		);
	GlobalConfiguration_typ : 	STRUCT
		machineIdentity : PM_MachineIdentity_typ;
	END_STRUCT;
	PM_MachineIdentity_typ : 	STRUCT
		factoryName : STRING[40]; (*ex: HQ, VulcanOne, ...*)
		machineNumber : UINT; (*ex: 0=invalid, 1..N (repeat in each factory)*)
		machineName : STRING[40]; (*ex: BETA, GEN2, DP1, DP2, DP3...*)
	END_STRUCT;
END_TYPE
```

### Global.var - Global variables
```iecst
VAR
	gMachineState : Machine_typ;
	gConfiguration : GlobalConfiguration_typ;
END_VAR
```

### MachineControl.typ
```iecst
(********************************************************************
 * COPYRIGHT -- Automation Resources Group
 ********************************************************************
 * Package: MachineControl
 * File: MachineControl.typ
 * Author: David Blackburn
 * Created: November 10, 2011
 ********************************************************************
 * Data types of package MachineControl
 ********************************************************************)

TYPE
	MachineAlarms_type : 	STRUCT
		components : vfAlarms_Component_typ;
		configuration : MachineAlarms_Configuration_type;
		commandStatus : ARRAY[0..9]OF STRING[80];
		messageStatus : STRING[80];
		MACHINE_ALARM : vfAlarms_Instance_type;
		REFERENCE_REQUIRED : vfAlarms_Instance_type;
		PERMMEM_DATA_RESTORED : vfAlarms_Instance_type;
		PERMMEM_FILE_ERROR : vfAlarms_Instance_type;
		PERMMEM_PERSISTER_ERROR : vfAlarms_Instance_type;
		PERMMEM_PERSISTER_SIZE_CHANGED : vfAlarms_Instance_type;
		SPLIT_CONFIG_LOAD_FAIL : vfAlarms_Instance_type;
		PERMMEM_PERSISTER_DATA_INVALID : vfAlarms_Instance_type;
		FILE_LINK_ERROR : vfAlarms_Instance_type;
		AUTOMATION_FAIL : vfAlarms_Instance_type;
		AUTOMATION_FAIL_COMMAND : vfAlarms_Instance_type;
		PACKML_STOP : vfAlarms_Instance_type;
		PACKML_ABORT : vfAlarms_Instance_type;
		AUTOMATION_CHECK_FAIL : vfAlarms_Instance_type;
	END_STRUCT;
	MachineAlarms_Configuration_type : 	STRUCT
		MACHINE_CONFIG_ALARM : STRING[80];
	END_STRUCT;
	SUBSTATES :
		(
		SUB_STATE_INIT,
		SUB_STATE_RESET_DRIVE_ERRORS,
		SUB_BOOTING_INIT_FILE_DEVICES,
		SUB_STATE_BOOTING_PERM_DATA,
		SUB_STATE_BOOTING_POSITION_CTRL,
		SUB_STATE_BOOTING_MOTION_FILTERS,
		SUB_STATE_BOOTING_WAIT_FOR_HOME,
		SUB_STATE_BOOTING_CLEAR_VIRT_REF,
		SUB_STATE_BOOTING_SW_LIMITS1,
		SUB_STATE_BOOTING_SW_LIMITS2,
		SUB_STATE_BOOTING_WAIT_FOR_PSU,
		SUB_STATE_STARTING_CHECK_REF,
		SUB_STATE_STARTING_SET_LIMITS,
		SUB_STATE_RESETTING_RESET_SAFETY,
		SUB_STATE_RESETTING_HOPPER,
		SUB_STATE_PSU_POWER,
		SUB_STATE_SERVO_POWER_GROUP1,
		SUB_STATE_SERVO_DEPOWER_GROUP1,
		SUB_STATE_SERVO_POWER_GROUP2,
		SUB_STATE_SERVO_DEPOWER_GROUP2,
		SUB_STATE_SERVO_POWER_GROUP3,
		SUB_STATE_SERVO_DEPOWER_GROUP3,
		SUB_STATE_SERVO_POWER_ALL,
		SUB_STATE_SERVO_HOME,
		SUB_STATE_SERVO_HOME_DONE,
		SUB_STATE_GEAR_IN,
		SUB_STATE_CHECK_CHILLER,
		SUB_STATE_CHECK_HOME,
		SUB_STATE_SERVO_PROMPT,
		SUB_STATE_GH_RECOVER,
		SUB_STATE_GH_MOVE_GANTRY,
		SUB_STATE_GANTRY_PROMPT,
		SUB_STATE_GANTRY_PARK,
		SUB_STATE_RECOATER_PROMPT,
		SUB_STATE_RECOATER_PARK,
		SUB_STATE_CONFIRM_PUMPS_WANTED,
		SUB_STATE_RESETTING_START_PUMPS,
		SUB_STATE_CONFIRM_LASERS_WANTED,
		SUB_STATE_RESETTING_LASERS_ON,
		SUB_STATE_START_SFC,
		SUB_STATE_EXITING_INIT,
		SUB_STATE_EXITING_CLEANUP,
		SUB_STATE_STOPPING_STOP_CNC,
		SUB_STATE_CLEARING_PROMPT_USER,
		SUB_STATE_CLEARING_START_PROGRAM,
		SUB_STATE_CLEARING_WAIT_FINISH,
		SUB_STATE_DISABLE_AXIS_ENAGAGE,
		SUB_STATE_SERVO_STOP,
		SUB_STATE_SERVO_POWER_OFF,
		SUB_STATE_PSU_POWER_OFF,
		SUB_STATE_BACKUP_HOME_DATA,
		SUB_STATE_STOP_DISABLE_MOTORS,
		SUB_STATE_DEPOWER_LASERS,
		SUB_STATE_STOP_PUMPS
		);
END_TYPE
```

### MachineControl.var
```iecst
(********************************************************************
 * COPYRIGHT -- Automation Resources Group
 ********************************************************************
 * Package: MachineControl
 * File: MachineControl.var
 * Author: David Blackburn
 * Created: November 10, 2011
 ********************************************************************
 * Variables of package MachineControl
 ********************************************************************)
VAR
	gMachine : Piper_typ := (0);
END_VAR
VAR RETAIN
	BootTime : TIME;
END_VAR
VAR
	gActiveMode : MODE_MACHINE_ENUM := MODE_MACHINE_AUTO;
	gRequestedMode : MODE_MACHINE_ENUM := MODE_MACHINE_AUTO;
	gMachineAlarms : MachineAlarms_type; (*General Alarms*)
END_VAR
```

### Program Logical/MachineControl/MachineMode/MachineMode (IEC)

#### PiperModule.var
```iecst
(********************************************************************
 * COPYRIGHT --
 ********************************************************************
 * Program: PiperModuleTemplate
 * File: PiperModuleTemplate.var
 * Author: Josh
 * Created: October 03, 2013
 ********************************************************************
 * Local variables of program PiperModuleTemplate
 ********************************************************************)
VAR
	ModuleInterface : Module_Interface_typ;
	Module : Piper_Module_Fub;
	piperCommands : task_command_type;
	_piperCommands : task_command_type;
END_VAR
```

### SafeLogicTypes.typ
```iecst
TYPE
	IO_SafeLOGIC_typ : 	STRUCT
		Status : IO_SL_Status_typ;
		Command : IO_SL_Commands_typ;
		Override : IO_SL_Override_typ;
		NonSafeInputs : IO_SL_NonSafeInputs_typ;
		SafeModuleOK : ARRAY[0..16]OF BOOL;
	END_STRUCT;
	IO_SL_Status_typ : 	STRUCT
		SafetyProgramRevision : UINT;
		SafetySystemReady : BOOL;
		EStopPressed : BOOL;
		GuardOpen_LoadZone : BOOL;
		GuardOpen_Airlock : BOOL;
		GuardOpen_Exterior : BOOL;
		GuardOpen_PrintZone : BOOL;
		SafetyReset_EStops : BOOL;
		SafetyReset_Guards_LoadZone : BOOL;
		SafetyReset_Guards_Pod : BOOL;
		SafetyReset_Guards_Airl : BOOL;
		SafetyReset_Guards_PrintZone : BOOL;
		SafetyReset_Lasers : BOOL;
		HeaterContactorEnabled : BOOL;
		AxesEnabled_Gantry : BOOL;
		AxesEnabled_Recoater : BOOL;
		AxesEnabled_Shuttle_AirLocks : BOOL;
		AxesEnabled_ZLifts : BOOL;
		RecoaterStepperEnabled : BOOL;
		RecoaterElectrodeEnabled : BOOL;
		SupplyEnabled_CDA : BOOL;
		SupplyEnabled_Argon : BOOL;
		ArgonSupplyEnabled_PrintZone : BOOL;
		ArgonEnabled_OBox_DShield : BOOL;
		ArgonEnabled_GasHead : BOOL;
		CDAEnabled_GasHead : BOOL;
		FBK_Error_EStop : BOOL;
		FBK_Error_Guard : BOOL;
		FBK_Error_Pneumatic : BOOL;
		FBK_Error_Heater : BOOL;
		FBK_Error_Drive : BOOL;
		FBK_Error_RecStepper : BOOL;
		FBK_Error_RecElectrode : BOOL;
		FBK_Error_Laser : BOOL;
		FBK_Error_VFLCR_LaserEDM : BOOL;
		FBK_Diag_EStop : UINT;
		FBK_Diag_Guard : UINT;
		FBK_Diag_Pneumatic : UINT;
		FBK_Diag_Heater : UINT;
		FBK_Diag_Drive : UINT;
		FBK_Diag_RecStepper : UINT;
		FBK_Diag_RecElectrode : UINT;
		FBK_Diag_Laser : UINT;
		FBK_Diag_VFLCR_LaserEDM0 : UINT;
		FBK_Diag_VFLCR_LaserEDM1 : UINT;
		FBK_Diag_VFLCR_LaserEDM2 : UINT;
		FBK_Diag_VFLCR_LaserEDM3 : UINT;
		LaserSafetyPwrContactRackError : ARRAY[0..6]OF BOOL;
		AirlockSealed_Right : BOOL;
		ExteriorLoadZoneInterlocked : BOOL;
		PodPresentSealed_Right : BOOL;
	END_STRUCT;
	IO_SL_Commands_typ : 	STRUCT
		RequestMachineSafetyReset : BOOL;
		RequestLaserSafetyReset : BOOL;
		RequestReleaseReset : BOOL;
		RequestUnlock_LoadZone : BOOL;
		RequestUnlock_PrintZone : BOOL;
		EnableHeaterContactor : BOOL;
		EnableLaserSafetyInterlock : BOOL;
		EnableAxes_Gantry : BOOL;
		EnableAxes_Recoater : BOOL;
		EnableAxes_Shuttle_Airlocks : BOOL;
		EnableAxes_ZLifts : BOOL;
		EnableRecoaterStepper : BOOL;
		EnableRecoaterElectrode : BOOL;
		EnablePneumaticsSupply : BOOL;
		EnableArgonSupply_PrintZonePurge : BOOL;
		SelectArgon_OBox_DShield : BOOL;
		SelectArgon_GasHead : BOOL;
		SelectCDA_GasHead : BOOL;
		RacksEnabled : UINT;
		RequestToEnterExteriorLoadZone : BOOL;
	END_STRUCT;
	IO_SL_NonSafeInputs_typ : 	STRUCT
		ArgonPreRegulatorPressureOK : BOOL;
		ArgonSupplyPressureOK : BOOL;
		CDASupplyPressureOK : BOOL;
		RequestExteriorZoneUnlock : BOOL;
		AcceleratedAirPurgeActive : BOOL;
	END_STRUCT;
	IO_SL_Override_typ : 	STRUCT
		Override_LoadZoneGuards : BOOL;
		Override_PrintZoneGuards : BOOL;
		Override_ControlStationEStop : BOOL;
		Override_SafetyLockoutBoxEStop : BOOL;
		Override_MachineMezEStop : BOOL;
		Override_MachineRearEStop : BOOL;
		Override_GasDistributionEStop : BOOL;
		Override_AirlockSafetyInterl : BOOL;
	END_STRUCT;
	IO_SDI_DUAL_typ : 	STRUCT
		CH1 : BOOL;
		CH2 : BOOL;
		DUAL_EVAL : BOOL;
		SAFEOK : BOOL;
	END_STRUCT;
	IO_SDO_DUAL_typ : 	STRUCT
		CH1 : BOOL;
		CH2 : BOOL;
		CH1_SAFEOK : BOOL;
		CH2_SAFEOK : BOOL;
	END_STRUCT;
	IO_SDI_SINGLE_typ : 	STRUCT
		CH1 : BOOL;
		SAFEOK : BOOL;
	END_STRUCT;
	IO_SDO_SINGLE_typ : 	STRUCT
		CH1 : BOOL;
		SAFEOK : BOOL;
	END_STRUCT;
END_TYPE
```

### Types.typ
```iecst
TYPE
	testCommand_typ : 	STRUCT
		induceLowSupplyPressure : BOOL;
		initAirPressure : BOOL;
		initNoEstopPressed : BOOL;
		induceOpenHatch : BOOL;
		induceEStopPressed : BOOL;
	END_STRUCT;
	test_typ : 	STRUCT
		command : testCommand_typ;
	END_STRUCT;
	IO_typ : 	STRUCT
		safeLOGIC : IO_SafeLOGIC_typ;
		DI_SafetyResetButton : ARRAY[0..1]OF BOOL;
		DO_InhibitAlarm_O2SafetyBox : BOOL;
		DO_SafetyResetLamp : BOOL;
		SDI_EStopButton_HandHeld : IO_SDI_DUAL_typ;
		SDI_EStop_LaserControlRoom : IO_SDI_DUAL_typ;
		DoorInterlock2 : IO_SD_Interlock_typ;
		DoorInterlock1 : IO_SD_Interlock_typ;
		SDI_SafetyLockoutSwitchMCC : IO_SDI_DUAL_typ;
		LaserSystem : ARRAY[0..MACHINE_MAI_LASER_RACKS]OF IO_SD_LaserSafety_typ;
		Chiller2TemperatureOK : BOOL;
		Chiller1TemperatureOK : BOOL;
		Chiller1Running : BOOL;
		Chiller2Running : BOOL;
		ChillerRunning : BOOL;
		SafetyStatus : BOOL;
		BatOBFlow : BOOL;
	END_STRUCT;
	Configuration_typ : 	STRUCT
		Exists : BOOL;
	END_STRUCT;
	localInterfaceCommand_typ : 	STRUCT
		resetAllSafety : BOOL;
		resetMachineSafety : BOOL;
		resetLaserSafety : BOOL;
	END_STRUCT;
	localInterfaceInternal_typ : 	STRUCT
		PLCOpen : AtnPlcOpenStatus;
		previousState : STATE;
		newCommand : BOOL;
		localLockout : BOOL;
		fbResetLaserOnPulse : VF_COMMON_PulseTrain;
		fbPulseBlueResetIndicator : VF_COMMON_PulseTrain;
		fbResetMachineOnPulse : VF_COMMON_PulseTrain;
		subSystemStatus : ARRAY[0..10]OF STRING[80];
		_safetyResetButton : BOOL;
		eStopIndex : USINT;
		interlockIndex : USINT;
		overrideIndex : USINT;
		resetAllSafety : AtnPLCOpen;
		ns_PodGaurdClosed : BOOL;
		ns_PigtailGaurdClosed : BOOL;
		alarmExteriorUnlock : BOOL;
		preventExteriorUnlock : BOOL;
		safetyTimeout : TON;
		interlocksOpen : BOOL;
		_interlocksOpen : BOOL;
	END_STRUCT;
	localInterfaceStatus_typ : 	STRUCT
		ready : BOOL;
		state : STATE;
		sequence : SEQUENCE;
		statusMessage : STRING[vfALARMS_MAX_SNIPPET_STR_LENGTH];
		allSafetyReset : BOOL;
		IOState : IOSTATE;
		eStopStatus : ARRAY[0..10]OF STRING[80];
		eStopStatusBool : BOOL;
		interlockStatus : ARRAY[0..10]OF STRING[80];
		interlockStatusBool : BOOL;
		overrideStatus : ARRAY[0..10]OF STRING[80];
		overrideStatusBool : BOOL;
		debrisShieldStatus : STRING[40];
		allActiveEStopOverridden : BOOL;
	END_STRUCT;
	localInterface_typ : 	STRUCT
		command : localInterfaceCommand_typ;
		status : localInterfaceStatus_typ;
		internal : localInterfaceInternal_typ;
	END_STRUCT;
	SEQUENCE :
		(
		SEQUENCE_IDLE,
		SEQUENCE_DONE,
		SEQUENCE_ERROR,
		SEQUENCE_EXECUTE_SAFETY_RESET,
		SEQUENCE_RESET_MACHINE_SAFETY,
		SEQUENCE_WAITING_FOR_MACH_SAFETY,
		SEQUENCE_RESET_LASER_SAFETY,
		SEQUENCE_WAITING_FOR_LSR_SAFETY
		);
	IOSTATE :
		(
		ENABLE_ARGON_PZ_PURGE,
		DISABLE_ARGON_PZ_PURGE,
		PURGE_GAS_HEAD_ARGON,
		PURGE_GAS_HEAD_CDA
		);
	STATE :
		(
		STATE_NOT_READY,
		STATE_READY,
		STATE_DONE,
		STATE_ERROR,
		STATE_RESET_MACHINE_SAFETY,
		STATE_RESET_LASER_SAFETY,
		STATE_RESET_ALL_SAFETY
		);
END_TYPE
```

### Types.typ
```iecst
TYPE
	MessageHandler_typ : 	STRUCT
		msgId : BOOL;
		ok : BOOL;
		cancel : BOOL;
	END_STRUCT;
	SFCControlApi_type : 	STRUCT
		command : SFCControlCommand_type;
		status : SFCControlStatus_type;
		inhibit : SFCControlInhibits_type;
		systems : STRING[80];
	END_STRUCT;
	SFCControlCommand_type : 	STRUCT
		pause : STRING[80];
		unpause : STRING[80];
		reset : STRING[80];
	END_STRUCT;
	SFCControlStatus_type : 	STRUCT
		sfc : STRING[80];
		sOMSModeActive : STRING[80];
		sOMSTestComplete : STRING[80];
	END_STRUCT;
	SFCControlInhibits_type : 	STRUCT
		_ : STRING[80];
	END_STRUCT;
	SFCControlDataApi_type : {REDUND_UNREPLICABLE} 	STRUCT
		pPause : REFERENCE TO BOOL;
		pBypass : REFERENCE TO BOOL;
		pTransition : REFERENCE TO BOOL;
		pSingleStep : REFERENCE TO BOOL;
	END_STRUCT;
	Automations_type : 	STRUCT
		command : AutomationsCommand_type;
		status : AutomationsStatus_type;
	END_STRUCT;
	AutomationsCommand_type : 	STRUCT
		recoat : STRING[80];
		scrape : STRING[80];
		refillHopper : STRING[80];
		printLayer : STRING[80];
		cleanGasHead : STRING[80];
		refillBuffer : STRING[80];
		refillOverheadHopper : STRING[80];
		initiateDoor : STRING[80];
		closeDoor : STRING[80];
		initiatePod : STRING[80];
	END_STRUCT;
	AutomationsStatus_type : 	STRUCT
		autonomousModeActive : STRING[80];
	END_STRUCT;
	MODE_MACHINE_ENUM :
		(
		MODE_MACHINE_AUTO,
		MODE_MACHINE_MANUAL_PROGRAM,
		MODE_MACHINE_MANUAL_JOG
		);
END_TYPE
```

### Variables.var
```iecst
VAR
	gSFCControlApi : SFCControlApi_type;
	gAutomations : Automations_type;
END_VAR
```

### Program Logical/Automation/SFCControl (IEC)

#### Main.st - Init, cyclic, exit code
```iecst
PROGRAM _INIT
	(* Insert code here *)

END_PROGRAM

PROGRAM _CYCLIC
	// Call PiperModuleInterface to interface with the rest of the machine
	PiperModuleInterface;

	//Call Fubs

	//The pause command must be set false. The current ATN commands are only set true,
	//This allows us to manually set the pause bits false as we need to
	anyPaused := FALSE;
	FOR index := 0 TO stateCount( gSFCControlApi.status.sfc ) DO
		IF forStateGetPointer( gSFCControlApi.status.sfc, index, 0, ADR(pSFCData), ADR(sSFCData) ) THEN
			dSFCData ACCESS pSFCData;
			dPause ACCESS dSFCData.pPause;
			dBypass ACCESS dSFCData.pBypass;
			dTrans ACCESS dSFCData.pTransition;
			dSingleStep ACCESS dSFCData.pSingleStep;

			IF dSingleStep AND NOT dPause AND dTrans THEN
				dPause := TRUE;
			END_IF

			IF task.internal.unpause.Execute OR task.internal.reset.Execute THEN
				dPause := FALSE;
			END_IF

			dBypass := dPause AND task.status.paused;
			anyPaused := anyPaused OR dPause;

		END_IF
	END_FOR

	task.internal.unpause.Command := gSFCControlApi.command.unpause;
	task.internal.unpause();
	task.internal.unpause.Execute := FALSE;

	task.internal.reset.Command := gSFCControlApi.command.reset;
	task.internal.reset();
	task.internal.reset.Execute := FALSE;

END_PROGRAM

PROGRAM _EXIT
	(* Insert code here *)

END_PROGRAM
```

#### Types.typ - Local data types
```iecst
TYPE
	localInterface_typ : 	STRUCT
		command : localInterfaceCommand_typ;
		parameters : localInterfaceParameter_typ;
		status : localInterfaceStatus_typ;
		internal : localInterfaceInternal_typ;
	END_STRUCT;
	localInterfaceCommand_typ : 	STRUCT
		stop : BOOL;
		_ : BOOL;
	END_STRUCT;
	localInterfaceParameter_typ : 	STRUCT
		_ : USINT;
	END_STRUCT;
	localInterfaceStatus_typ : 	STRUCT
		ErrorState : STRING[80];
		paused : BOOL;
	END_STRUCT;
	localInterfaceInternal_typ : 	STRUCT
		PLCOpen : AtnPlcOpenStatus;
		unpause : AtnPLCOpen;
		reset : AtnPLCOpen;
	END_STRUCT;
END_TYPE
```

#### Variables.var - Local variables
```iecst
VAR
	task : localInterface_typ;
	index : INT;
	pPause : {REDUND_UNREPLICABLE} UDINT;
	dPause : REFERENCE TO BOOL;
	sPause : UDINT;
	pSFCData : UDINT;
	sSFCData : UDINT;
	dSFCData : REFERENCE TO SFCControlDataApi_type;
	dBypass : REFERENCE TO BOOL;
	anyPaused : BOOL;
	dTrans : REFERENCE TO BOOL;
	dSingleStep : REFERENCE TO BOOL;
END_VAR
```

#### PiperInterface.st
```iecst
(********************************************************************
 * COPYRIGHT --
 ********************************************************************
 * Program: MachineProg
 * File: PiperModuleInterface.st
 * Author: Josh
 * Created: October 03, 2013
 ********************************************************************
 * Implementation of program MachineProg
 ********************************************************************)

ACTION PiperModuleInterface:

	//Give this module a name so it is easier to debug
	ModuleInterface.ModuleName:=	'SFC Control';

	//Add a module to the Piper
	Module.ModuleInterface:=	ADR(ModuleInterface);
	Module.Piper:= 	ADR(gMachine);
	Module();

	task.status.paused := FALSE;

	// Handle any machine states that this module needs to respond to
	CASE ModuleInterface.PiperState OF
		//		MACH_ST_BOOTING:
		//		MACH_ST_CLEARING:
		//		MACH_ST_STOPPED:
		//		MACH_ST_STARTING:
		//		MACH_ST_IDLE:
		//		MACH_ST_SUSPENDED:
		MACH_ST_EXECUTE:
			IF anyPaused THEN
				task.status.paused := TRUE;
				ModuleInterface.ModuleResponse:=	MACH_ST_NOT_READY;
			ELSE
				task.status.paused := FALSE;
				ModuleInterface.ModuleResponse:=	ModuleInterface.PiperState;
			END_IF
		//		MACH_ST_ABORTING:
		//		MACH_ST_ABORTED:
		//		MACH_ST_HOLDING:
		//		MACH_ST_HELD:
		MACH_ST_STOPPING,
		MACH_ST_ABORTING:
			task.internal.reset.Execute := TRUE;
			IF task.internal.reset.Done
			OR task.internal.reset.Error
			OR task.internal.reset.Aborted THEN

				ModuleInterface.ModuleResponse:=	ModuleInterface.PiperState;

			END_IF

		MACH_ST_UNHOLDING,
		MACH_ST_SUSPENDING:

			task.internal.unpause.Execute := TRUE;
			IF task.internal.unpause.Done THEN

				ModuleInterface.ModuleResponse:=	ModuleInterface.PiperState;

			ELSIF task.internal.unpause.Error OR task.internal.unpause.Aborted THEN

				gMachine.IN.CMD.Stop := TRUE;

	//			vfAlarmEdgeSnippet( gMachineAlarms.components, gMachineAlarms.PACKML_STOP, 'Stop due to unpause failure');

				logInfo( 'App', 0, 'Stop due to failure to unpause', 0 );

			END_IF
		//		MACH_ST_UNSUSPENDING:
		//		MACH_ST_RESETTING:
		//		MACH_ST_COMPLETING:
		//		MACH_ST_COMPLETE:
		MACH_ST_BYPASSED:

		ELSE
			ModuleInterface.ModuleResponse:=	ModuleInterface.PiperState;

	END_CASE

END_ACTION
```

### Program Logical/Automation/SFCCommon (IEC)

#### Types.typ - Local data types
```iecst
(*
This is a template for the SFC types
*)

TYPE
	Configuration_typ : 	STRUCT
		errorAborts : BOOL;
	END_STRUCT;
	localInterface_typ : 	STRUCT
		command : localInterfaceCommand_typ;
		parameters : localInterfaceParameter_typ;
		status : localInterfaceStatus_typ;
		internal : localInterfaceInternal_typ;
	END_STRUCT;
	localInterfaceCommand_typ : 	STRUCT
		stop : BOOL;
		_ : BOOL;
	END_STRUCT;
	localInterfaceParameter_typ : 	STRUCT
		_ : USINT;
	END_STRUCT;
	localInterfaceStatus_typ : 	STRUCT
		activeOperation : STRING[80];
		activeStep : USINT;
		statusMessage : STRING[vfALARMS_MAX_SNIPPET_STR_LENGTH];
		statusID : UDINT;
		subSystemStatus : ARRAY[0..9]OF STRING[80];
		ready : BOOL;
		ErrorState : STRING[80];
	END_STRUCT;
	localInterfaceInternal_typ : 	STRUCT
		PLCOpen : AtnPlcOpenStatus;
		newCommand : BOOL;
	END_STRUCT;
END_TYPE
```

#### Action.st
```iecst
//Continuous action connected to step one
ACTION FunctionblockCalls:
	// Data collection info updated for the event

	task.status.activeStep := SFCCurrentStep;

	IF task.command.stop THEN
		SFCReset := 		TRUE;
		Command.Execute := 	FALSE;
		Command();
	ELSE
		SFCReset := 		FALSE;
	END_IF

	IF Command.Aborted THEN

		logStateChange_0.StateName := CONCAT(Command.Command, ' - Aborted');
		task.status.statusID := ERR_FUB_REDUNDANT;
		task.internal.PLCOpen.status := ERR_FUB_REDUNDANT;
		task.status.ErrorState := SFCCurrentStep;

//		AlarmText := CONCAT(logStateChange_0.ModuleName, ' Step: ');
//		AlarmText := CONCAT(AlarmText, SFCCurrentStep);
//		gMachineAlarms.commandStatus := Command.StatusMessage;
//		gMachineAlarms.messageStatus := task.status.statusMessage;
//		vfAlarmEdgeSnippet( gMachineAlarms.components, gMachineAlarms.AUTOMATION_FAIL_COMMAND, AlarmText);

		SFCReset := 		TRUE;
		Command.Execute := 	FALSE;
		Command();

		logStateChange_0.State := logStateChange_0.State + 1;

	ELSIF Command.Error THEN

		logStateChange_0.StateName := CONCAT(Command.Command, ' - Error');
		task.status.statusID := Command.Status;
		task.internal.PLCOpen.status := Command.Status;
		task.status.ErrorState := SFCCurrentStep;

//		AlarmText := CONCAT(logStateChange_0.ModuleName, ' Step: ');
//		AlarmText := CONCAT(AlarmText, SFCCurrentStep);
//		gMachineAlarms.commandStatus := Command.StatusMessage;
//		gMachineAlarms.messageStatus := task.status.statusMessage;
//		vfAlarmEdgeSnippet( gMachineAlarms.components, gMachineAlarms.AUTOMATION_FAIL_COMMAND, AlarmText);

		SFCReset := 		TRUE;
		Command.Execute := 	FALSE;
		Command();

		logStateChange_0.State := logStateChange_0.State + 1;

	ELSIF StepError THEN

		StepError := FALSE;

		logStateChange_0.StateName := CONCAT(SFCCurrentStep, ' - Error');
		//		task.status.statusID := this should be set by the erroring state;
		task.internal.PLCOpen.status := 	ERR_FUB_ENABLE_FALSE;
		task.status.ErrorState := SFCCurrentStep;

//		AlarmText := CONCAT(logStateChange_0.ModuleName, ' Step: ');
//		AlarmText := CONCAT(AlarmText, SFCCurrentStep);
//		AlarmText := CONCAT(AlarmText, ' (Step Error)');
//		gMachineAlarms.commandStatus := Command.StatusMessage;
//		gMachineAlarms.messageStatus := task.status.statusMessage;
//		vfAlarmEdgeSnippet( gMachineAlarms.components, gMachineAlarms.AUTOMATION_FAIL, AlarmText);

		SFCReset := 		TRUE;
		Command.Execute := 	FALSE;
		Command();

		logStateChange_0.State := logStateChange_0.State + 1;

	ELSE

		IF logStateChange_0.StateName <> SFCCurrentStep THEN
			logStateChange_0.State := logStateChange_0.State + 1;
		END_IF
		logStateChange_0.StateName := SFCCurrentStep;
	END_IF

	Command.pParameters := 0;
	Command.sParameters := 0;

	logStateChange_0.LoggerName:= 'App';
	ST_name( 0, ADR(logStateChange_0.ModuleName), ADR(group) );
	logStateChange_0();

	//	StepDone := FALSE;
	//	StepRetry := FALSE;

	IF NOT startStepActive AND _startStepActive THEN

		task.status.statusID := ERR_FUB_BUSY;
		task.status.ErrorState := '';
		task.status.statusMessage := '';

	END_IF

	_startStepActive := startStepActive;
	startStepActive := FALSE;

END_ACTION

//Action running during step1
ACTION Step1Active:

	logStateChange_0.State := 0;

	//If Step 1 is active, clear out any old fub statuses
	IF Command.Busy OR Command.Done OR Command.Aborted OR Command.Error THEN
		Command.Execute := 	FALSE;
		Command();
	END_IF

	//If we get here and have a busy status, it means we completed succefully
	IF NOT _startStepActive THEN
		IF task.status.statusID = ERR_FUB_BUSY THEN
			task.status.statusID := ERR_OK;
			task.internal.PLCOpen.status := ERR_OK;
		ELSE
			task.internal.PLCOpen.status := task.status.statusID;
		END_IF
	END_IF

	StepDone := FALSE;
	StepError := FALSE;

	IF messageHandler.msgId <> 0 THEN
		messageHandler.msgId := 0;
		MessageBox_RemoveMsg( messageHandler.msgId );
	END_IF

	startStepActive := TRUE;

END_ACTION
```

#### Common.var - Local variables
```iecst
VAR
	group : USINT;
	sfcData : SFCControlDataApi_type;
	task : {REDUND_UNREPLICABLE} localInterface_typ;
	SFCReset : BOOL;
	SFCTrans : BOOL;
	SFCPause : BOOL;
	SFCCurrentStep : STRING[80];
	SFCSingleStep : BOOL;
	OK : BOOL;
	StepError : BOOL;
	CycleDone : BOOL;
	StepDoneOpenLayer : BOOL;
	StepDone : BOOL;
	StepContinue : BOOL;
	StepRetry : BOOL;
	StepPopExit : BOOL;
	startStepActive : BOOL;
	_startStepActive : BOOL;
	logStateChange_0 : logStateChange;
	ModuleInterface : Module_Interface_typ;
	Module : Piper_Module_Fub;
END_VAR
VAR RETAIN
	Configuration : Configuration_typ;
END_VAR
VAR
	init : BOOL;
	messageHandler : MessageHandler_typ;
	AlarmText : STRING[vfALARMS_MAX_SNIPPET_STR_LENGTH];
	StepExit : BOOL;
	ScanTaken : BOOL;
END_VAR
```

#### PiperInterface.st
```iecst
ACTION PiperModuleInterface:

	IF NOT init THEN
		init:= TRUE;

		//Subscribe the SFC commands so they can be controled externally
		subscribeCommandBool(gSFCControlApi.command.reset, logStateChange_0.ModuleName, SFCReset);
		subscribeCommandBool(gSFCControlApi.command.pause, logStateChange_0.ModuleName, SFCPause);

		//We need to register the SFCPause bit as a parameter so it can be written to false, currently commands only write true.
		registerStateParameters(gSFCControlApi.status.sfc, logStateChange_0.ModuleName, ADR(sfcData), SIZEOF(sfcData));
	END_IF
	sfcData.pBypass := ADR(ModuleInterface.ModuleBypass);
	sfcData.pPause := ADR(SFCPause);
	sfcData.pTransition := ADR(SFCTrans);
	sfcData.pSingleStep := ADR(SFCSingleStep);

	//Give this module a name so it is easier to debug
	ModuleInterface.ModuleName:=	logStateChange_0.ModuleName;

	//Add a module to the Piper
	Module.ModuleInterface:=	ADR(ModuleInterface);
	Module.Piper:= 	ADR(gMachine);
	Module();

	//Don't reset operations if we are bypassed, as this can mess with
	// The SFC while it's paused.
	//IF ModuleInterface.PiperState <> MACH_ST_BYPASSED THEN

	//	ResetOperation;

	//END_IF

	// Handle any machine states that this module needs to respond to
	CASE ModuleInterface.PiperState OF
		//		MACH_ST_BOOTING:
		//		MACH_ST_CLEARING:
		//		MACH_ST_STOPPED:
		MACH_ST_STARTING:

			CASE ModuleInterface.PiperSubState OF
				SUB_STATE_INIT:
					task.status.statusID := ERR_OK;
					ModuleInterface.ModuleSubStateRequest := SUB_STATE_START_SFC;

				SUB_STATE_START_SFC:

					SelectOperation;
					ModuleInterface.ModuleResponse:=	ModuleInterface.PiperState;

			END_CASE

			//		MACH_ST_IDLE:
			//		MACH_ST_SUSPENDED:
		MACH_ST_EXECUTE:

			IF task.status.statusID = ERR_OK THEN

				ModuleInterface.ModuleResponse:=	ModuleInterface.PiperState;

			ELSIF task.status.statusID = ERR_FUB_BUSY THEN

				ModuleInterface.ModuleResponse :=	MACH_ST_NOT_READY;

			ELSE

				IF Configuration.errorAborts THEN
					IF ModuleInterface.ModuleResponse <> MACH_ST_ERROR THEN
						ModuleInterface.ModuleResponse:=	MACH_ST_ERROR;
					//	vfAlarmEdgeSnippet( gMachineAlarms.components, gMachineAlarms.PACKML_ABORT, logStateChange_0.ModuleName);
					END_IF
				ELSE

					IF NOT gMachine.IN.CMD.Stop THEN

				//		vfAlarmEdgeSnippet( gMachineAlarms.components, gMachineAlarms.PACKML_STOP, logStateChange_0.ModuleName);
						logInfo( 'App', UDINT_TO_UINT(task.status.statusID), 'Stop due to SFC status', 0 );
						gMachine.IN.CMD.Stop := TRUE;

					END_IF

				END_IF
			END_IF

		MACH_ST_STOPPING:
			SFCReset := TRUE;
			// SOMS abort handskake handling

			IF (gMachineState._previousOperation = MACH_OP_OMS_TEST ) AND stateAnyFalse( gSFCControlApi.status.sOMSTestComplete , TRUE ) AND stateAnyTrue( gVFLCR.status.usingGen3LaserCalibrationApp , TRUE )
				AND stateAllTrue(gSFCControlApi.status.sOMSModeActive,FALSE) AND stateAllTrue(gVFLCR.status.heartbeatLaserCalibrationAppOk,FALSE) THEN
				executeCommand(gVFLCR.command.passAbortedHandshakeWithoutAck);
			END_IF

			gMachineState._previousOperation := MACH_OP_NONE;

			ModuleInterface.ModuleResponse:=	ModuleInterface.PiperState;

		MACH_ST_ABORTING:

			SFCReset := TRUE;
			// SOMS abort handskake handling

			IF (gMachineState._previousOperation = MACH_OP_OMS_TEST ) AND stateAnyFalse( gSFCControlApi.status.sOMSTestComplete , TRUE ) AND stateAnyTrue( gVFLCR.status.usingGen3LaserCalibrationApp , TRUE )
				AND stateAllTrue(gSFCControlApi.status.sOMSModeActive,FALSE) AND stateAllTrue(gVFLCR.status.heartbeatLaserCalibrationAppOk,FALSE) THEN
				executeCommand(gVFLCR.command.passAbortedHandshakeWithoutAck);
			END_IF

			gMachineState._previousOperation := MACH_OP_NONE;

			ModuleInterface.ModuleResponse:=	ModuleInterface.PiperState;

			IF messageHandler.msgId <> 0 THEN
				messageHandler.msgId := 0;
				MessageBox_RemoveMsg( messageHandler.msgId );
			END_IF

		MACH_ST_HOLDING:
			SFCPause := TRUE;
			ModuleInterface.ModuleResponse:=	ModuleInterface.PiperState;

		MACH_ST_UNHOLDING:
			//At this point the task is paused, so this actually isn't really a case to handle here.
			// Unpause happens externally in SFCControl Task.
			SFCPause := FALSE;
			ModuleInterface.ModuleResponse:=	ModuleInterface.PiperState;

			//		MACH_ST_ABORTED:
			//		MACH_ST_HELD:
			//		MACH_ST_SUSPENDING:
			//		MACH_ST_UNSUSPENDING:
			//		MACH_ST_RESETTING:
			//		MACH_ST_COMPLETING:
			//		MACH_ST_COMPLETE:

		MACH_ST_BYPASSED:

		ELSE
			ModuleInterface.ModuleResponse:=	ModuleInterface.PiperState;

	END_CASE

//	ModuleInterface.ModuleBypass := SFCPause;

	brsmemset( ADR(task.command), 0, SIZEOF(task.command));

END_ACTION
```

#### commands.st
```iecst
ACTION SelectOperation:

	(* EACH SFC should impliment a select operation action*)

END_ACTION

ACTION ResetOperation:

	(* EACH SFC should impliment a reset operation action*)

END_ACTION
```

### Program Logical/Automation/DataDistributionSFC (IEC)

#### Cyclic.sfc - Cyclic code
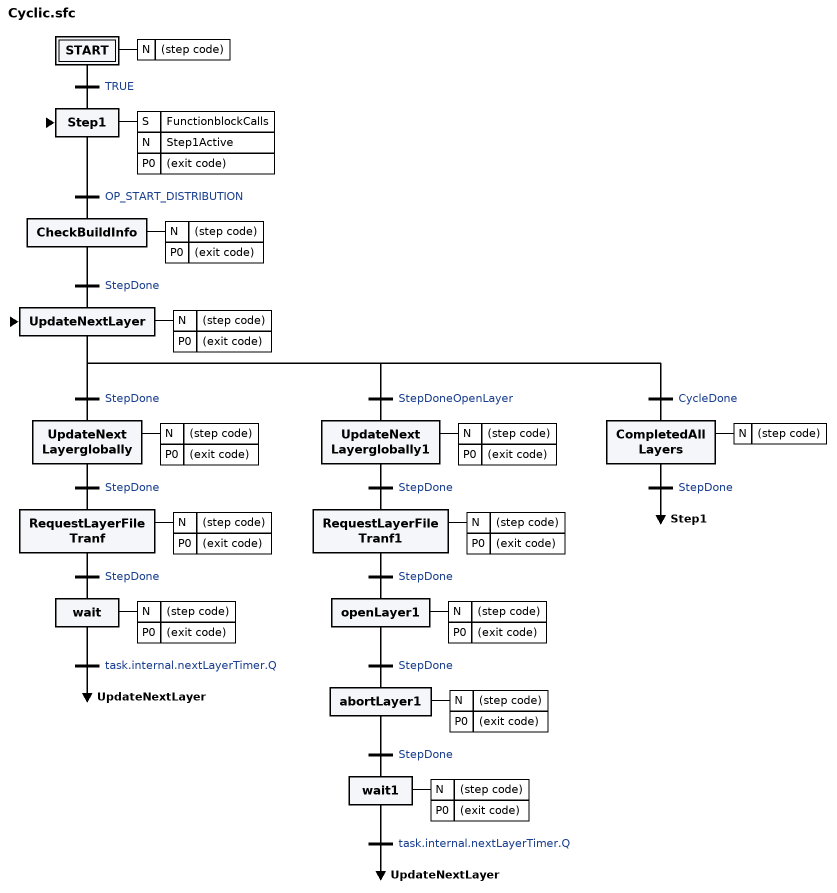
```iecst
PROGRAM _CYCLIC
INITIAL_STEP START:

SFCReset := FALSE;
END_STEP
TRANSITION FROM START TO Step1:=
TRUE
END_TRANSITION
IEC_STEP Step1:
FunctionblockCalls(S);
Step1Active(N);
END_STEP
EXIT_ACTION
task.internal.completedLayers := FALSE;
task.internal.completedCycles := 0;

END_ACTION
TRANSITION FROM Step1 TO CheckBuildInfo:=
OP_START_DISTRIBUTION
END_TRANSITION
STEP CheckBuildInfo:

gPrintJobManagement.currentState.currentLayerNumber := 1;
IF gPrintJobManagement.currentState.buildInfoCheckValid THEN
	StepDone := TRUE;
ELSE
	//TODO:	task.status.statusID := SOME_ERROR;
	StepError := TRUE;
END_IF
END_STEP
EXIT_ACTION
StepDone := FALSE;
END_ACTION
TRANSITION FROM CheckBuildInfo TO UpdateNextLayer:=
StepDone
END_TRANSITION
STEP UpdateNextLayer:
task.internal.nextLayerNumber  := gPrintJobManagement.currentState.currentLayerNumber + 1;

// Incrementing to the next layer is only permitted as long as the last layer has yet to be printed.
IF ( task.internal.nextLayerNumber <= gPrintJobManagement.currentState.numberOfLayers ) AND gPrintJobManagement.currentState.openAndCloseLayers THEN

	StepDoneOpenLayer := TRUE;

ELSIF ( task.internal.nextLayerNumber <= gPrintJobManagement.currentState.numberOfLayers ) THEN

	StepDone := TRUE;

ELSE

	task.internal.completedCycles := task.internal.completedCycles + 1;
	CycleDone := TRUE;

	task.status.statusMessage := 'Invalid Next layer';

	//Can't print the requested layer, since it isn't the next layer
	//vfAlarmEdge( gPrintJobManagement.alarms.components, gPrintJobManagement.alarms.InvalidCurrentLayer_AL0026 );

END_IF
END_STEP
EXIT_ACTION
StepDone := FALSE;
StepDoneOpenLayer := FALSE;
CycleDone := FALSE;
(* TODO: Insert Program *)
END_ACTION
TRANSITION FROM UpdateNextLayer TO UpdateNextLayerglobally:=
StepDone
END_TRANSITION
TRANSITION FROM UpdateNextLayer TO UpdateNextLayerglobally1:=
StepDoneOpenLayer
END_TRANSITION
STEP UpdateNextLayerglobally1:
gPrintJobManagement.currentState.nextLayerNumber := task.internal.nextLayerNumber;
gPrintJobManagement.currentState.currentLayerNumber := gPrintJobManagement.currentState.nextLayerNumber;

StepDone := TRUE;

END_STEP
EXIT_ACTION
StepDone := FALSE;
END_ACTION
TRANSITION FROM UpdateNextLayerglobally1 TO RequestLayerFileTranf1:=
StepDone
END_TRANSITION
STEP RequestLayerFileTranf1:

buildDistCommand.Command := gBuildDistributorApi.commands.distributeLayerFile;
buildDistCommand.Execute := TRUE;
buildDistCommand();

IF buildDistCommand.Done OR  gPrintJobManagement.status.distributionLayerComplete OR (gOpcData_FromBuildPC.CurrentDistributionLayer = gOpcData_ToBuildPC.CurrentPrintLayer) THEN

	StepDone := TRUE;
	gPrintJobManagement.status.distributionLayerComplete := FALSE;
	buildDistCommand.Execute := FALSE;
	buildDistCommand();
ELSIF buildDistCommand.Error OR buildDistCommand.Aborted THEN

	StepDone := FALSE;
	StepError := TRUE;
	buildDistCommand.Execute := FALSE;
	buildDistCommand();

END_IF
END_STEP
EXIT_ACTION
StepDone := FALSE;
END_ACTION
TRANSITION FROM RequestLayerFileTranf1 TO openLayer1:=
StepDone
END_TRANSITION
STEP openLayer1:
Command.Command :=  gVFLCR.command.openLayer;
//TODO: VALIDATE THIS  IS CORRECT!
openLayerParameters.parameters.selectedBuildLayout :=	gPrintJobManagement.currentState.buildLayout;
openLayerParameters.parameters.selectedLayer :=			gPrintJobManagement.currentState.currentLayerNumber;
openLayerParameters.parameters.selectedPrintNumber :=	gPrintJobManagement.currentState.printNumber;
Command.pParameters := ADR(openLayerParameters);
Command.sParameters := SIZEOF(openLayerParameters);
Command.Execute := TRUE;
Command();
IF Command.Done THEN
	StepDone := TRUE;
	Command.Execute := FALSE;
	Command();
ELSE
	StepDone := FALSE;
END_IF
END_STEP
EXIT_ACTION
StepDone := FALSE;
END_ACTION
TRANSITION FROM openLayer1 TO abortLayer1:=
StepDone
END_TRANSITION
STEP abortLayer1:
Command.Command :=  gVFLCR.command.abortLayer;
Command.Execute := TRUE;
Command();
IF Command.Done THEN
	StepDone := TRUE;
	Command.Execute := FALSE;
	Command();
ELSE
	StepDone := FALSE;
END_IF

END_STEP
EXIT_ACTION
StepDone := FALSE;
END_ACTION
TRANSITION FROM abortLayer1 TO wait1:=
StepDone
END_TRANSITION
STEP wait1:
task.internal.nextLayerTimer.PT := T#5s;
task.internal.nextLayerTimer.IN := TRUE;
task.internal.nextLayerTimer();

END_STEP
EXIT_ACTION
task.internal.nextLayerTimer.IN := FALSE;
task.internal.nextLayerTimer();
(* TODO: Insert Program *)
END_ACTION
TRANSITION FROM wait1 TO UpdateNextLayer:=
task.internal.nextLayerTimer.Q
END_TRANSITION
(* @SFCISJUMP := 'UpdateNextLayer' *)
TRANSITION FROM UpdateNextLayer TO CompletedAllLayers:=
CycleDone
END_TRANSITION
STEP CompletedAllLayers:
//task.internal.completedLayers := TRUE;

//IF task.command.closePopup THEN

	//task.internal.completedLayers := FALSE;
StepDone := TRUE;
gPrintJobManagement.currentState.currentLayerNumber := 0;

//END_IF
END_STEP
TRANSITION FROM CompletedAllLayers TO Step1:=
StepDone
END_TRANSITION
(* @SFCISJUMP := 'Step1' *)
STEP UpdateNextLayerglobally:
gPrintJobManagement.currentState.nextLayerNumber := task.internal.nextLayerNumber;
gPrintJobManagement.currentState.currentLayerNumber := gPrintJobManagement.currentState.nextLayerNumber;

StepDone := TRUE;

END_STEP
EXIT_ACTION
StepDone := FALSE;
END_ACTION
TRANSITION FROM UpdateNextLayerglobally TO RequestLayerFileTranf:=
StepDone
END_TRANSITION
STEP RequestLayerFileTranf:

buildDistCommand.Command := gBuildDistributorApi.commands.distributeLayerFile;
buildDistCommand.Execute := TRUE;
buildDistCommand();

IF buildDistCommand.Done OR  gPrintJobManagement.status.distributionLayerComplete OR (gOpcData_FromBuildPC.CurrentDistributionLayer = gOpcData_ToBuildPC.CurrentPrintLayer) THEN

	StepDone := TRUE;
	gPrintJobManagement.status.distributionLayerComplete := FALSE;
	buildDistCommand.Execute := FALSE;
	buildDistCommand();
ELSIF buildDistCommand.Error OR buildDistCommand.Aborted THEN

	StepDone := FALSE;
	StepError := TRUE;
	buildDistCommand.Execute := FALSE;
	buildDistCommand();

END_IF
END_STEP
EXIT_ACTION
StepDone := FALSE;
END_ACTION
TRANSITION FROM RequestLayerFileTranf TO wait:=
StepDone
END_TRANSITION
STEP wait:
task.internal.nextLayerTimer.PT := T#5s;
task.internal.nextLayerTimer.IN := TRUE;
task.internal.nextLayerTimer();

END_STEP
EXIT_ACTION
task.internal.nextLayerTimer.IN := FALSE;
task.internal.nextLayerTimer();
(* TODO: Insert Program *)
END_ACTION
TRANSITION FROM wait TO UpdateNextLayer:=
task.internal.nextLayerTimer.Q
END_TRANSITION
(* @SFCISJUMP := 'UpdateNextLayer' *)
END_PROGRAM
```

#### Types.typ - Local data types
```iecst
TYPE
	Configuration_typ : 	STRUCT
		errorAborts : BOOL;
	END_STRUCT;
	localInterfaceCommand_typ : 	STRUCT
		closePopup : BOOL;
		stop : BOOL;
		_ : BOOL;
	END_STRUCT;
	localInterfaceInternal_typ : 	STRUCT
		PLCOpen : AtnPlcOpenStatus;
		nextLayerTimer : TON;
		nextLayerNumber : UINT;
		completedCycles : UINT;
		completedLayers : BOOL;
		newCommand : BOOL;
	END_STRUCT;
	localInterfaceStatus_typ : 	STRUCT
		activeOperation : STRING[80];
		activeStep : STRING[80];
		statusMessage : STRING[vfALARMS_MAX_SNIPPET_STR_LENGTH];
		subSystemStatus : ARRAY[0..9]OF STRING[80];
		ready : BOOL;
		ErrorState : STRING[80];
		statusID : UDINT;
	END_STRUCT;
	localInterface_typ : 	STRUCT
		command : localInterfaceCommand_typ;
		status : localInterfaceStatus_typ;
		internal : localInterfaceInternal_typ;
	END_STRUCT;
END_TYPE
```

#### Variables.var - Local variables
```iecst
VAR
	Command : AtnPLCOpenWithParameters;
	OP_START_DISTRIBUTION : BOOL;
	OP_ABORT_DISTRIBUTION : BOOL;
	buildDistCommand : AtnPLCOpenWithParameters;
	openLayerParameters : VFLCROpenLayerCommandPars_typ;
END_VAR
```

- Common.var (reference to Logical/Automation/SFCCommon/Common.var)

- PiperInterface.st (reference to Logical/Automation/SFCCommon/PiperInterface.st)

- Action.st (reference to Logical/Automation/SFCCommon/Action.st)

#### commands.st
```iecst
ACTION SelectOperation:

	CASE gMachineState.operation  OF

		MACH_OP_START_DISTRIBUTION:
			OP_START_DISTRIBUTION := TRUE;
			task.status.statusID := 	ERR_FUB_BUSY;
			task.status.activeOperation:= 'Distribution Started';

		MACH_OP_ABORT_DISTRIBUTION:
			OP_ABORT_DISTRIBUTION := TRUE;
			task.status.statusID := 	ERR_FUB_BUSY;
			task.status.activeOperation:= 'Distribution Aborted';

	END_CASE

END_ACTION

ACTION ResetOperation:

	OP_START_DISTRIBUTION := FALSE;
	OP_ABORT_DISTRIBUTION := FALSE;

END_ACTION
```

### Program Logical/Automation/LaserGen3SFC
